// TwinCAT 3 PLC project SDSM3
// Title: SDS M2
// Company: Aperture Science
// Author: A. Wallace
// ProjectVersion: 2.6.1
// ProgramVersion: 3.1.0.9
// libraries:
//   LCLSVacuumLib, * (SLAC)
//   Tc2_Standard, * (Beckhoff Automation GmbH)
//   Tc2_System, * (Beckhoff Automation GmbH)
//   Tc3_Module, * (Beckhoff Automation GmbH)
//   LCLS General,0.1.2,SLAC
//   Tc2_EtherCAT,3.3.7.0,Beckhoff Automation GmbH
//   Tc2_IoFunctions,3.3.8.0,Beckhoff Automation GmbH
//   Tc2_MC2,3.3.15.0,Beckhoff Automation GmbH
//   Tc2_ModbusSrv,3.3.1.0,Beckhoff Automation GmbH
//   Tc2_SerialCom,3.3.6.0,Beckhoff Automation GmbH
//   Tc2_SUPS,3.3.4.0,Beckhoff Automation GmbH
//   Tc2_Utilities,3.3.17.0,Beckhoff Automation GmbH
// project tree:
//   DUTs/ALI/ E_AxisMoveMode.TcDUT (not stored), E_CTRL_MODE.TcDUT, E_PropValveFBState.TcDUT (not stored), HMI_PropValveCtrlState.TcDUT, ST_ALI.TcDUT, ST_ManipAxis.TcDUT, ST_PIDParams.TcDUT, ST_PressureController.TcDUT, ST_PropValveMKS253.TcDUT
//   DUTs/Bronkhorst/ E_BHElFlowUnit.TcDUT (not stored), ST_BhElFlow.TcDUT, ST_BhFMControl.TcDUT, ST_BhFMStatus.TcDUT
//   DUTs/ E_AxisMotionState.TcDUT, ST_M3GasManifold.TcDUT, ST_ManifoldValve.TcDUT (not stored), ST_Proportionair.TcDUT, ST_RegDeadbandControls.TcDUT (not stored), ST_Regulator.TcDUT (not stored), ST_Selector.TcDUT, ST_SelectorM3.TcDUT (not stored), ST_SensirionFM.TcDUT (not stored), ST_Shaker.TcDUT (not stored), ST_ShakerControls.TcDUT
//   DUTs/IO_Structs/ ST_ALIIO.TcDUT, ST_M2SelectorIO.TcDUT, ST_M3DeviceBaseIO.TcDUT (not stored), ST_M3GasManifoldIO.TcDUT (not stored), ST_M3PressCtrlIO.TcDUT (not stored), ST_M3SelectorIO.TcDUT
//   DUTs/Sensirion/ ST_SensirionFMControl.TcDUT, ST_SensirionFMStatus.TcDUT
//   DUTs/TEC/ ST_TECControl.TcDUT (not stored), ST_TECStatus.TcDUT (not stored)
//   DUTs/Vici/ ST_ViciControl.TcDUT, ST_ViciStatus.TcDUT (not stored)
//   GVLs/ GVL.TcGVL, GVL_Autosave.TcGVL, GVL_ComBuffers.TcGVL, GVL_Devices.TcGVL, GVL_IO.TcGVL, GVL_misc.TcGVL (not stored)
//   / PlcTask.TcTTO, SerialComm.TcTTO (not stored)
//   POUs/ALI/ FB_ALI.TcPOU, FB_PID_EXT.TcPOU, MC_SmoothMover.TcPOU, F_AxisRef_To_MSTA.TcPOU, FB_ManipAxis.TcPOU, FB_PropValve.TcPOU
//   POUs/Bronkhorst/ FB_L01Driver.TcPOU, FB_FlowBusTransaction.TcPOU (not stored)
//   POUs/ FB_SelectorM3.TcPOU, MAIN.TcPOU, p_ALI.TcPOU, p_Autosave.TcPOU, p_AutoWash.TcPOU, p_CoolerShaker.TcPOU, p_ESTOP.TcPOU, p_Manifold.TcPOU, p_ModbusRx.TcPOU, p_ModbusTx.TcPOU, p_Regulators.TcPOU, p_SampleSelector.TcPOU (not stored), p_SampleSelector2.TcPOU (not stored), p_Shakers.TcPOU, p_SoftIO.TcPOU, p_VacGaugeSup.TcPOU, SerialTxRx.TcPOU, p_StatusLights.TcPOU
//   POUs/Helpers/ FB_EcatDiag.TcPOU (not stored), FB_ManiValve.TcPOU (not stored), FB_SelectorSync.TcPOU, FB_ShiftByteArray.TcPOU
//   POUs/Regulators/ FB_ProportionairRegulator.TcPOU, FB_Regulator.TcPOU, F_rPressure.TcPOU (not stored)
//   POUs/Sensirion/ FB_SensirionDriver.TcPOU, FB_SensirionTransaction.TcPOU (not stored), fSHDLCChecksum.TcPOU (not stored)
//   POUs/TEC/ FB_TECDriver.TcPOU, FB_TECTransaction.TcPOU (not stored)
//   POUs/VICI/ FB_ViciDriver.TcPOU, FB_ViciTransaction.TcPOU
//   Version/ Global_Version.TcGVL
//   VISUs/ Main.TcVIS (not stored)
// real-time tasks:
//   TASK SerialComm: cycle T#5ms, priority 1, ADS port 350
//   TASK PlcTask: cycle T#10ms, priority 20, ADS port 351
// motion (NC):
//   TASK NC-Task 1 SAF: cycle T#2ms, priority 4, ADS port 501
//   TASK NC-Task 1 SVB: cycle T#10ms, priority 8, ADS port 511
//   AXIS ALI_X (id 3)
//     Dynamic: AccelerationMaximum=300, DecelerationMaximum=300, Acceleration=100, Deceleration=100
//     Velo: Maximum=5
//     PositionAreaControl: Range=0.005, RefSync=0.005
//     TargetPosControl: Range=0.0001
//     OtherSettings: AllowMotionCmdToSlave=true
//     encoder EncType=4
//       EncPara: ScaleFactorNumerator=0.001, MaxCount=#x0000ffff
//         Inc: RefSoftSyncMask=#x0000ffff
//     drive DrvType=24
//       Analog: VeloReferenz=12.7
//       TimeComp: TaskDelayCycles=1
//     controller CtrType=1
//       CtrPara: PriorControlFactor=1
//         PosDiffControl: Range=1
//         Observer: BandWidth=20
//   AXIS ALI_Z (id 5)
//     Dynamic: AccelerationMaximum=1000, DecelerationMaximum=1000, Acceleration=10, Deceleration=10, Jerk=100, DelayTime=0.08
//     Velo: Maximum=1
//     OtherSettings: AllowMotionCmdToSlave=true
//     encoder EncType=4
//       EncPara: ScaleFactorNumerator=3.96875e-005, MaxCount=#x0000ffff
//         Inc: RefSoftSyncMask=#x0000ffff
//     drive DrvType=24
//       Analog: VeloReferenz=5.08
//       TimeComp: TaskDelayCycles=1
//     controller CtrType=1
//       CtrPara: PriorControlFactor=1
//         PosDiffControl: Enable=false
//         Observer: BandWidth=20
//   AXIS ALI_Y (id 4)
//     Dynamic: DelayTime=0.08
//     Velo: Maximum=5
//     PositionAreaControl: Range=0.005, RefSync=0.005
//     TargetPosControl: Range=0.0001
//     OtherSettings: AllowMotionCmdToSlave=true
//     encoder EncType=4
//       EncPara: ScaleFactorNumerator=0.001, MaxCount=#x0000ffff
//         Inc: RefSoftSyncMask=#x0000ffff
//     drive DrvType=24
//       Analog: VeloReferenz=12.7
//       TimeComp: TaskDelayCycles=1
//     controller CtrType=1
//       CtrPara: PriorControlFactor=1
//         PosDiffControl: Range=1.5
//         Observer: BandWidth=20
//   AXIS ALI_PropValve (id 6)
//     General: UnitName=°
//     OtherSettings: AllowMotionCmdToSlave=true
//     encoder EncType=4
//       EncPara: ScaleFactorNumerator=0.028125, MaxCount=#x0000ffff
//         SoftEndMinControl: Enable=true
//         SoftEndMaxControl: Enable=true, Range=2900
//         Inc: RefSoftSyncMask=#x0000ffff
//     drive DrvType=24
//       Analog: VeloReferenz=3600
//       TimeComp: TaskDelayCycles=1
//     controller CtrType=1
//       CtrPara: PriorControlFactor=1
//         Observer: BandWidth=20
// I/O:
//   DEVICE MAIN (EtherCAT), AmsNetId 5.35.66.22.2.1
//     Term 1 (EK1200) [EK1200-5000 EtherCAT Power supply (2A E-Bus)]
//       Term 14 (EL3064) [EL3064 4Ch. Ana. Input 0-10V] (disabled)
//       Term 23 (EL4004) [EL4004 4Ch. Ana. Output 0-10V, 12bit] (disabled)
//       Term 25 (EL1124) [EL1124 4Ch. Dig. Input 5V, 10µs, Sensor Power] (disabled)
//       Term 17 (EL1008) [EL1008 8Ch. Dig. Input 24V, 3ms] (disabled)
//       Term 18 (EL2008) [EL2008 8Ch. Dig. Output 24V, 0.5A] (disabled)
//       Term 19 (EL2798) [EL2798 8Ch. Dig. Output 24V AC/DC, 2A, potential-free] (disabled)
//       Term 24 (EK1110) [EK1110 EtherCAT extension]
//     SC2 (EP9128-0021) [EP9128-0021 8x EtherCAT junction]
//       Box 32 (EP9128-1021) [EP9128-1021 8x EtherCAT junction - Dev A]
//       Box 33 (EP9128-2021) [EP9128-2021 8x EtherCAT junction - Dev B]
//     SC1 (EP9128-0021) [EP9128-0021 8x EtherCAT junction] (disabled)
//       Box 29 (EP9128-1021) [EP9128-1021 8x EtherCAT junction - Dev A]
//       Box 30 (EP9128-2021) [EP9128-2021 8x EtherCAT junction - Dev B]
//     SC3 (EP9128-0021) [EP9128-0021 8x EtherCAT junction] (disabled)
//       Box 21 (EP9128-1021) [EP9128-1021 8x EtherCAT junction - Dev A]
//       Box 22 (EP9128-2021) [EP9128-2021 8x EtherCAT junction - Dev B]
//     ALI (EP1111) [EP1111-0000 ID-Switch]
//     ALI_X (EP7041-0002) [EP7041-0002 1Ch. Stepper motor output stage (50V, 5A)]
//     ALI_Y (EP7041-0002) [EP7041-0002 1Ch. Stepper motor output stage (50V, 5A)]
//     ALI_Z (EP7041-0002) [EP7041-0002 1Ch. Stepper motor output stage (50V, 5A)]
//     ALI_X_ENC (EP5101-0011) [EP5101-0011 1Ch. Inc. Encoder 5V, D-SUB15]
//     ALI_Gauges (EP3174-0002) [EP3174-0002 4Ch. Ana. Input +/-10V, 0-10V, 0/4-20mA configurable]
//     ALI_PropValve (EP7041-0002) [EP7041-0002 1Ch. Stepper motor output stage (50V, 5A)]
//     ALI_Y_ENC (EP5101-0011) [EP5101-0011 1Ch. Inc. Encoder 5V, D-SUB15]
//     ALI_DIO (EP2338-0001) [EP2338-0001 8 Ch. Dig. Input/Output 24V, 0,5A, M8] (disabled)
//     M2 Selector A (EP1111) [EP1111-0000 ID-Switch]
//     M2 Selector A (EP6002-0002) [EP6002-0002 Interface (RS232/422/485)]
//     M2 Selector A (EP2338-0001) [EP2338-0001 8 Ch. Dig. Input/Output 24V, 0,5A, M8]
//     M2 Selector B (EP1111) [EP1111-0000 ID-Switch]
//     M2 Selector B (EP6002-0002) [EP6002-0002 Interface (RS232/422/485)]
//     M2 Selector B (EP2338-0001) [EP2338-0001 8 Ch. Dig. Input/Output 24V, 0,5A, M8]
//     M3 Selector A (EP1111) [EP1111-0000 ID-Switch]
//     M3 Selector A Digital IO (EP2338-1001) [EP2338-1001 8 Ch. Dig. Input/Output 24V, 3ms, 0,5A, M8]
//     M3 Selector A Serial IO (EP6002-0002) [EP6002-0002 Interface (RS232/422/485)]
//     M3 Selector A Mass Flow Meter (Mass Flow / Pressure Controller - Slave) [Mass Flow / Pressure Controller - Slave]
//     M3 Selector B (EP1111) [EP1111-0000 ID-Switch]
//     M3 Selector B Digital IO (EP2338-1001) [EP2338-1001 8 Ch. Dig. Input/Output 24V, 3ms, 0,5A, M8]
//     M3 Selector B Serial IO (EP6002-0002) [EP6002-0002 Interface (RS232/422/485)]
//     M3 Selector B Mass Flow Meter (Mass Flow / Pressure Controller - Slave) [Mass Flow / Pressure Controller - Slave]
//     PCM A (EP1111) [EP1111-0000 ID-Switch]
//     PCM A (EP4374-0002) [EP4374-0002 2Ch. Ana. Input +/-10V, 0-10V, 0/4-20mA configurable; 2Ch. Ana. Output +/-10V, 0-10V, 0/4-20mA configurable]
//     PCM A (EP3174-0002) [EP3174-0002 4Ch. Ana. Input +/-10V, 0-10V, 0/4-20mA configurable]
//     PCM A (EP6002-0002) [EP6002-0002 Interface (RS232/422/485)]
//     PCM B (EP1111) [EP1111-0000 ID-Switch]
//     PCM B (EP4374-0002) [EP4374-0002 2Ch. Ana. Input +/-10V, 0-10V, 0/4-20mA configurable; 2Ch. Ana. Output +/-10V, 0-10V, 0/4-20mA configurable]
//     PCM B (EP3174-0002) [EP3174-0002 4Ch. Ana. Input +/-10V, 0-10V, 0/4-20mA configurable] (disabled)
//     PCM B (EP6002-0002) [EP6002-0002 Interface (RS232/422/485)] (disabled)
//     Gas_Mani (EP1111) [EP1111-0000 ID-Switch]
//     Gas_Mani_NeedleValve (EP4374-0002) [EP4374-0002 2Ch. Ana. Input +/-10V, 0-10V, 0/4-20mA configurable; 2Ch. Ana. Output +/-10V, 0-10V, 0/4-20mA configurable]
//     Gas_Mani_ValveCtrl (EP2338-0001) [EP2338-0001 8 Ch. Dig. Input/Output 24V, 0,5A, M8]
//     Gas_Mani_ValveRbk (EP2338-0001) [EP2338-0001 8 Ch. Dig. Input/Output 24V, 0,5A, M8]
// variable links:
//   NC-Task 1 SAF/Axes/ALI_PropValve <-> MAIN (EtherCAT)/ALI_PropValve (EP7041-0002)
//     Drive/Inputs/In/nState1 @bit 3 <-> STM Status/Status/Error
//     Drive/Inputs/In/nState1 @bit 5 <-> STM Status/Status/Moving negative
//     Drive/Inputs/In/nState1 @bit 4 <-> STM Status/Status/Moving positive
//     Drive/Inputs/In/nState1 @bit 1 <-> STM Status/Status/Ready
//     Drive/Inputs/In/nState1 <-> STM Status/Status/Ready to enable
//     Drive/Inputs/In/nState1 @bit 6 <-> STM Status/Status/Torque reduced
//     Drive/Inputs/In/nState1 @bit 2 <-> STM Status/Status/Warning
//     Drive/Inputs/In/nState2 @bit 3 <-> STM Status/Status/Digital input 1
//     Drive/Inputs/In/nState2 @bit 4 <-> STM Status/Status/Digital input 2
//     Drive/Inputs/In/nState2 @bit 5 <-> STM Status/Status/Sync error
//     Drive/Inputs/In/nState2 @bit 7 <-> STM Status/Status/TxPDO Toggle
//     Drive/Inputs/In/nState4 @bit 1 <-> WcState/InputToggle
//     Drive/Inputs/In/nState4 <-> WcState/WcState
//     Drive/Outputs/Out/nCtrl1 <-> STM Control/Control/Enable
//     Drive/Outputs/Out/nCtrl1 @bit 2 <-> STM Control/Control/Reduce torque
//     Drive/Outputs/Out/nCtrl1 @bit 1 <-> STM Control/Control/Reset
//     Drive/Outputs/Out/nCtrl2 @bit 3 <-> STM Control/Control/Digital output 1
//     Drive/Outputs/Out/nDataOut2[0] <-> STM Velocity/Velocity
//     Enc/Inputs/In/nDataIn1[0] <-> ENC Status compact/Counter value
//     Enc/Inputs/In/nDataIn2[0] <-> ENC Status compact/Latch value
//     Enc/Inputs/In/nState1 @bit 4 <-> ENC Status compact/Status/Counter overflow
//     Enc/Inputs/In/nState1 @bit 3 <-> ENC Status compact/Status/Counter underflow
//     Enc/Inputs/In/nState1 @bit 7 <-> ENC Status compact/Status/Extrapolation stall
//     Enc/Inputs/In/nState1 <-> ENC Status compact/Status/Latch C valid
//     Enc/Inputs/In/nState1 @bit 1 <-> ENC Status compact/Status/Latch extern valid
//     Enc/Inputs/In/nState1 @bit 2 <-> ENC Status compact/Status/Set counter done
//     Enc/Inputs/In/nState2 @bit 4 <-> ENC Status compact/Status/Status of extern latch
//     Enc/Inputs/In/nState2 <-> ENC Status compact/Status/Status of input A
//     Enc/Inputs/In/nState2 @bit 1 <-> ENC Status compact/Status/Status of input B
//     Enc/Inputs/In/nState2 @bit 2 <-> ENC Status compact/Status/Status of input C
//     Enc/Inputs/In/nState2 @bit 5 <-> ENC Status compact/Status/Sync error
//     Enc/Inputs/In/nState2 @bit 7 <-> ENC Status compact/Status/TxPDO Toggle
//     Enc/Inputs/In/nState4 @bit 1 <-> WcState/InputToggle
//     Enc/Inputs/In/nState4 <-> WcState/WcState
//     Enc/Outputs/Out/nCtrl1 <-> ENC Control compact/Control/Enable latch C
//     Enc/Outputs/Out/nCtrl1 @bit 3 <-> ENC Control compact/Control/Enable latch extern on negative edge
//     Enc/Outputs/Out/nCtrl1 @bit 1 <-> ENC Control compact/Control/Enable latch extern on positive edge
//     Enc/Outputs/Out/nCtrl1 @bit 2 <-> ENC Control compact/Control/Set counter
//     Enc/Outputs/Out/nDataOut1[0] <-> ENC Control compact/Set counter value
//   NC-Task 1 SAF/Axes/ALI_X <-> MAIN (EtherCAT)/ALI_X (EP7041-0002)
//     Drive/Inputs/In/nState1 @bit 3 <-> STM Status/Status/Error
//     Drive/Inputs/In/nState1 @bit 5 <-> STM Status/Status/Moving negative
//     Drive/Inputs/In/nState1 @bit 4 <-> STM Status/Status/Moving positive
//     Drive/Inputs/In/nState1 @bit 1 <-> STM Status/Status/Ready
//     Drive/Inputs/In/nState1 <-> STM Status/Status/Ready to enable
//     Drive/Inputs/In/nState1 @bit 6 <-> STM Status/Status/Torque reduced
//     Drive/Inputs/In/nState1 @bit 2 <-> STM Status/Status/Warning
//     Drive/Inputs/In/nState2 @bit 3 <-> STM Status/Status/Digital input 1
//     Drive/Inputs/In/nState2 @bit 4 <-> STM Status/Status/Digital input 2
//     Drive/Inputs/In/nState2 @bit 5 <-> STM Status/Status/Sync error
//     Drive/Inputs/In/nState2 @bit 7 <-> STM Status/Status/TxPDO Toggle
//     Drive/Inputs/In/nState4 @bit 1 <-> WcState/InputToggle
//     Drive/Inputs/In/nState4 <-> WcState/WcState
//     Drive/Outputs/Out/nCtrl1 <-> STM Control/Control/Enable
//     Drive/Outputs/Out/nCtrl1 @bit 2 <-> STM Control/Control/Reduce torque
//     Drive/Outputs/Out/nCtrl1 @bit 1 <-> STM Control/Control/Reset
//     Drive/Outputs/Out/nCtrl2 @bit 3 <-> STM Control/Control/Digital output 1
//     Drive/Outputs/Out/nDataOut2[0] <-> STM Velocity/Velocity
//   NC-Task 1 SAF/Axes/ALI_X <-> MAIN (EtherCAT)/ALI_X_ENC (EP5101-0011)
//     Enc/Inputs/In/nDataIn1[0] <-> ENC Status compact/Counter value
//     Enc/Inputs/In/nDataIn2[0] <-> ENC Status compact/Latch value
//     Enc/Inputs/In/nState1 @bit 4 <-> ENC Status compact/Status/Counter overflow
//     Enc/Inputs/In/nState1 @bit 3 <-> ENC Status compact/Status/Counter underflow
//     Enc/Inputs/In/nState1 @bit 7 <-> ENC Status compact/Status/Extrapolation stall
//     Enc/Inputs/In/nState1 <-> ENC Status compact/Status/Latch C valid
//     Enc/Inputs/In/nState1 @bit 1 <-> ENC Status compact/Status/Latch extern valid
//     Enc/Inputs/In/nState1 @bit 6 <-> ENC Status compact/Status/Open circuit
//     Enc/Inputs/In/nState1 @bit 2 <-> ENC Status compact/Status/Set counter done
//     Enc/Inputs/In/nState1 @bit 5 <-> ENC Status compact/Status/Status of input status
//     Enc/Inputs/In/nState2 @bit 4 <-> ENC Status compact/Status/Status of extern latch
//     Enc/Inputs/In/nState2 <-> ENC Status compact/Status/Status of input A
//     Enc/Inputs/In/nState2 @bit 1 <-> ENC Status compact/Status/Status of input B
//     Enc/Inputs/In/nState2 @bit 2 <-> ENC Status compact/Status/Status of input C
//     Enc/Inputs/In/nState2 @bit 3 <-> ENC Status compact/Status/Status of input gate
//     Enc/Inputs/In/nState4 @bit 1 <-> WcState/InputToggle
//     Enc/Inputs/In/nState4 <-> WcState/WcState
//     Enc/Outputs/Out/nCtrl1 <-> ENC Control compact/Control/Enable latch C
//     Enc/Outputs/Out/nCtrl1 @bit 3 <-> ENC Control compact/Control/Enable latch extern on negative edge
//     Enc/Outputs/Out/nCtrl1 @bit 1 <-> ENC Control compact/Control/Enable latch extern on positive edge
//     Enc/Outputs/Out/nCtrl1 @bit 2 <-> ENC Control compact/Control/Set counter
//     Enc/Outputs/Out/nDataOut1[0] <-> ENC Control compact/Set counter value
//   NC-Task 1 SAF/Axes/ALI_Y <-> MAIN (EtherCAT)/ALI_Y (EP7041-0002)
//     Drive/Inputs/In/nState1 @bit 3 <-> STM Status/Status/Error
//     Drive/Inputs/In/nState1 @bit 5 <-> STM Status/Status/Moving negative
//     Drive/Inputs/In/nState1 @bit 4 <-> STM Status/Status/Moving positive
//     Drive/Inputs/In/nState1 @bit 1 <-> STM Status/Status/Ready
//     Drive/Inputs/In/nState1 <-> STM Status/Status/Ready to enable
//     Drive/Inputs/In/nState1 @bit 6 <-> STM Status/Status/Torque reduced
//     Drive/Inputs/In/nState1 @bit 2 <-> STM Status/Status/Warning
//     Drive/Inputs/In/nState2 @bit 3 <-> STM Status/Status/Digital input 1
//     Drive/Inputs/In/nState2 @bit 4 <-> STM Status/Status/Digital input 2
//     Drive/Inputs/In/nState2 @bit 5 <-> STM Status/Status/Sync error
//     Drive/Inputs/In/nState2 @bit 7 <-> STM Status/Status/TxPDO Toggle
//     Drive/Inputs/In/nState4 @bit 1 <-> WcState/InputToggle
//     Drive/Inputs/In/nState4 <-> WcState/WcState
//     Drive/Outputs/Out/nCtrl1 <-> STM Control/Control/Enable
//     Drive/Outputs/Out/nCtrl1 @bit 2 <-> STM Control/Control/Reduce torque
//     Drive/Outputs/Out/nCtrl1 @bit 1 <-> STM Control/Control/Reset
//     Drive/Outputs/Out/nCtrl2 @bit 3 <-> STM Control/Control/Digital output 1
//     Drive/Outputs/Out/nDataOut2[0] <-> STM Velocity/Velocity
//   NC-Task 1 SAF/Axes/ALI_Y <-> MAIN (EtherCAT)/ALI_Y_ENC (EP5101-0011)
//     Enc/Inputs/In/nDataIn1[0] <-> ENC Status compact/Counter value
//     Enc/Inputs/In/nDataIn2[0] <-> ENC Status compact/Latch value
//     Enc/Inputs/In/nState1 @bit 4 <-> ENC Status compact/Status/Counter overflow
//     Enc/Inputs/In/nState1 @bit 3 <-> ENC Status compact/Status/Counter underflow
//     Enc/Inputs/In/nState1 @bit 7 <-> ENC Status compact/Status/Extrapolation stall
//     Enc/Inputs/In/nState1 <-> ENC Status compact/Status/Latch C valid
//     Enc/Inputs/In/nState1 @bit 1 <-> ENC Status compact/Status/Latch extern valid
//     Enc/Inputs/In/nState1 @bit 6 <-> ENC Status compact/Status/Open circuit
//     Enc/Inputs/In/nState1 @bit 2 <-> ENC Status compact/Status/Set counter done
//     Enc/Inputs/In/nState1 @bit 5 <-> ENC Status compact/Status/Status of input status
//     Enc/Inputs/In/nState2 @bit 4 <-> ENC Status compact/Status/Status of extern latch
//     Enc/Inputs/In/nState2 <-> ENC Status compact/Status/Status of input A
//     Enc/Inputs/In/nState2 @bit 1 <-> ENC Status compact/Status/Status of input B
//     Enc/Inputs/In/nState2 @bit 2 <-> ENC Status compact/Status/Status of input C
//     Enc/Inputs/In/nState2 @bit 3 <-> ENC Status compact/Status/Status of input gate
//     Enc/Inputs/In/nState4 @bit 1 <-> WcState/InputToggle
//     Enc/Inputs/In/nState4 <-> WcState/WcState
//     Enc/Outputs/Out/nCtrl1 <-> ENC Control compact/Control/Enable latch C
//     Enc/Outputs/Out/nCtrl1 @bit 3 <-> ENC Control compact/Control/Enable latch extern on negative edge
//     Enc/Outputs/Out/nCtrl1 @bit 1 <-> ENC Control compact/Control/Enable latch extern on positive edge
//     Enc/Outputs/Out/nCtrl1 @bit 2 <-> ENC Control compact/Control/Set counter
//     Enc/Outputs/Out/nDataOut1[0] <-> ENC Control compact/Set counter value
//   NC-Task 1 SAF/Axes/ALI_Z <-> MAIN (EtherCAT)/ALI_Z (EP7041-0002)
//     Drive/Inputs/In/nState1 @bit 3 <-> STM Status/Status/Error
//     Drive/Inputs/In/nState1 @bit 5 <-> STM Status/Status/Moving negative
//     Drive/Inputs/In/nState1 @bit 4 <-> STM Status/Status/Moving positive
//     Drive/Inputs/In/nState1 @bit 1 <-> STM Status/Status/Ready
//     Drive/Inputs/In/nState1 <-> STM Status/Status/Ready to enable
//     Drive/Inputs/In/nState1 @bit 6 <-> STM Status/Status/Torque reduced
//     Drive/Inputs/In/nState1 @bit 2 <-> STM Status/Status/Warning
//     Drive/Inputs/In/nState2 @bit 3 <-> STM Status/Status/Digital input 1
//     Drive/Inputs/In/nState2 @bit 4 <-> STM Status/Status/Digital input 2
//     Drive/Inputs/In/nState2 @bit 5 <-> STM Status/Status/Sync error
//     Drive/Inputs/In/nState2 @bit 7 <-> STM Status/Status/TxPDO Toggle
//     Drive/Inputs/In/nState4 @bit 1 <-> WcState/InputToggle
//     Drive/Inputs/In/nState4 <-> WcState/WcState
//     Drive/Outputs/Out/nCtrl1 <-> STM Control/Control/Enable
//     Drive/Outputs/Out/nCtrl1 @bit 2 <-> STM Control/Control/Reduce torque
//     Drive/Outputs/Out/nCtrl1 @bit 1 <-> STM Control/Control/Reset
//     Drive/Outputs/Out/nCtrl2 @bit 3 <-> STM Control/Control/Digital output 1
//     Drive/Outputs/Out/nDataOut2[0] <-> STM Velocity/Velocity
//     Enc/Inputs/In/nDataIn1[0] <-> ENC Status compact/Counter value
//     Enc/Inputs/In/nDataIn2[0] <-> ENC Status compact/Latch value
//     Enc/Inputs/In/nState1 @bit 4 <-> ENC Status compact/Status/Counter overflow
//     Enc/Inputs/In/nState1 @bit 3 <-> ENC Status compact/Status/Counter underflow
//     Enc/Inputs/In/nState1 @bit 7 <-> ENC Status compact/Status/Extrapolation stall
//     Enc/Inputs/In/nState1 <-> ENC Status compact/Status/Latch C valid
//     Enc/Inputs/In/nState1 @bit 1 <-> ENC Status compact/Status/Latch extern valid
//     Enc/Inputs/In/nState1 @bit 2 <-> ENC Status compact/Status/Set counter done
//     Enc/Inputs/In/nState2 @bit 4 <-> ENC Status compact/Status/Status of extern latch
//     Enc/Inputs/In/nState2 <-> ENC Status compact/Status/Status of input A
//     Enc/Inputs/In/nState2 @bit 1 <-> ENC Status compact/Status/Status of input B
//     Enc/Inputs/In/nState2 @bit 2 <-> ENC Status compact/Status/Status of input C
//     Enc/Inputs/In/nState2 @bit 5 <-> ENC Status compact/Status/Sync error
//     Enc/Inputs/In/nState2 @bit 7 <-> ENC Status compact/Status/TxPDO Toggle
//     Enc/Inputs/In/nState4 @bit 1 <-> WcState/InputToggle
//     Enc/Inputs/In/nState4 <-> WcState/WcState
//     Enc/Outputs/Out/nCtrl1 <-> ENC Control compact/Control/Enable latch C
//     Enc/Outputs/Out/nCtrl1 @bit 3 <-> ENC Control compact/Control/Enable latch extern on negative edge
//     Enc/Outputs/Out/nCtrl1 @bit 1 <-> ENC Control compact/Control/Enable latch extern on positive edge
//     Enc/Outputs/Out/nCtrl1 @bit 2 <-> ENC Control compact/Control/Set counter
//     Enc/Outputs/Out/nDataOut1[0] <-> ENC Control compact/Set counter value
//   SDSM3/SDSM3 Instance <-> MAIN (EtherCAT)
//     PlcTask Inputs/GVL.g_aEcatMaster1 <-> InfoData/AmsNetId
//     PlcTask Inputs/GVL_Devices.stALI.i_SyncUnitWC <-> SyncUnits/[ALI (EP1111)]/PlcTask/WcState/WcState
//     PlcTask Inputs/GVL_IO.iq_stM2SelectorA.i_SyncUnitWC <-> SyncUnits/[M2 Selector A (EP1111)]/PlcTask/WcState/WcState
//     PlcTask Inputs/GVL_IO.iq_stM3SelectorA.i_SyncUnitWC <-> SyncUnits/[M3 Selector A (EP1111)]/PlcTask/WcState/WcState
//     PlcTask Inputs/GVL_IO.iq_stM2SelectorB.i_SyncUnitWC <-> SyncUnits/[M2 Selector B (EP1111)]/<unreferenced>/WcState/WcState
//     PlcTask Inputs/GVL_IO.iq_stM3GasManifold.i_SyncUnitWC <-> SyncUnits/[Gas_Mani (EP1111)]/PlcTask/WcState/WcState
//     PlcTask Inputs/GVL_IO.iq_stM3SelectorB.i_SyncUnitWC <-> SyncUnits/[M3 Selector B (EP1111)]/PlcTask/WcState/WcState
//     PlcTask Inputs/GVL_IO.iq_stPressCtrlA.i_SyncUnitWC <-> SyncUnits/[PCM A (EP1111)]/PlcTask/WcState/WcState
//     PlcTask Inputs/GVL_IO.iq_stPressCtrlB.i_SyncUnitWC <-> SyncUnits/[PCM B (EP1111)]/PlcTask/WcState/WcState
//   SDSM3/SDSM3 Instance <-> MAIN (EtherCAT)/ALI_Gauges (EP3174-0002)
//     PlcTask Inputs/GVL_Devices.stALI.i_EP3174_Ch{1..4} <-> AI Standard Channel {1..4}/Value  (4 links)
//   SDSM3/SDSM3 Instance <-> MAIN (EtherCAT)/ALI_PropValve (EP7041-0002)
//     PlcTask Inputs/GVL_Devices.stALI.stPropVlv.i_HLS <-> STM Status/Status/Digital input 1
//     PlcTask Inputs/GVL_Devices.stALI.stPropVlv.i_LLS <-> STM Status/Status/Digital input 2
//   SDSM3/SDSM3 Instance <-> MAIN (EtherCAT)/ALI_X (EP7041-0002)
//     PlcTask Inputs/GVL_Devices.stALI.axisX.xHiLS <-> STM Status/Status/Digital input 2
//     PlcTask Inputs/GVL_Devices.stALI.axisX.xLoLS <-> STM Status/Status/Digital input 1
//   SDSM3/SDSM3 Instance <-> MAIN (EtherCAT)/ALI_Y (EP7041-0002)
//     PlcTask Inputs/GVL_Devices.stALI.axisY.xHiLS <-> STM Status/Status/Digital input 2
//     PlcTask Inputs/GVL_Devices.stALI.axisY.xLoLS <-> STM Status/Status/Digital input 1
//   SDSM3/SDSM3 Instance <-> MAIN (EtherCAT)/ALI_Z (EP7041-0002)
//     PlcTask Inputs/GVL_Devices.stALI.axisZ.xHiLS <-> STM Status/Status/Digital input 2
//     PlcTask Inputs/GVL_Devices.stALI.axisZ.xLoLS <-> STM Status/Status/Digital input 1
//   SDSM3/SDSM3 Instance <-> MAIN (EtherCAT)/Gas_Mani_NeedleValve (EP4374-0002)
//     PlcTask Inputs/GVL_IO.iq_stM3GasManifold.i_EP4374_Ch1 <-> AI Inputs Channel 1/Value
//     PlcTask Inputs/GVL_IO.iq_stM3GasManifold.i_EP4374_Ch2 <-> AI Inputs Channel 2/Value
//     PlcTask Outputs/GVL_IO.iq_stM3GasManifold.q_EP4374_Ch3 <-> AO Outputs Channel 3/Analog output
//     PlcTask Outputs/GVL_IO.iq_stM3GasManifold.q_EP4374_Ch4 <-> AO Outputs Channel 4/Analog output
//   SDSM3/SDSM3 Instance <-> MAIN (EtherCAT)/Gas_Mani_ValveCtrl (EP2338-0001)
//     PlcTask Outputs/GVL_IO.iq_stM3GasManifold.q_EP2338_Ch{1..8} <-> Channel {9..16}/Output  (8 links)
//   SDSM3/SDSM3 Instance <-> MAIN (EtherCAT)/Gas_Mani_ValveRbk (EP2338-0001)
//     PlcTask Inputs/GVL_IO.iq_stM3GasManifold.i_EP2338_Ch{1..8} <-> Channel {1..8}/Input  (8 links)
//   SDSM3/SDSM3 Instance <-> MAIN (EtherCAT)/M2 Selector A (EP2338-0001)
//     PlcTask Inputs/GVL_IO.iq_stM2SelectorA.i_EP2338_Ch{5..8} <-> Channel {5..8}/Input  (4 links)
//     PlcTask Outputs/GVL_IO.iq_stM2SelectorA.q_EP2338_Ch{1..4} <-> Channel {9..12}/Output  (4 links)
//   SDSM3/SDSM3 Instance <-> MAIN (EtherCAT)/M2 Selector A (EP6002-0002)
//     SerialComm Inputs/GVL_IO.iq_stM2SelectorA.stComIn_EP6002P1/D[0] <-> COM TxPDO-Map Inputs Channel 1/Data In 0
//     SerialComm Inputs/GVL_IO.iq_stM2SelectorA.stComIn_EP6002P1/D[10] <-> COM TxPDO-Map Inputs Channel 1/Data In 10
//     SerialComm Inputs/GVL_IO.iq_stM2SelectorA.stComIn_EP6002P1/D[11] <-> COM TxPDO-Map Inputs Channel 1/Data In 11
//     SerialComm Inputs/GVL_IO.iq_stM2SelectorA.stComIn_EP6002P1/D[12] <-> COM TxPDO-Map Inputs Channel 1/Data In 12
//     SerialComm Inputs/GVL_IO.iq_stM2SelectorA.stComIn_EP6002P1/D[13] <-> COM TxPDO-Map Inputs Channel 1/Data In 13
//     SerialComm Inputs/GVL_IO.iq_stM2SelectorA.stComIn_EP6002P1/D[14] <-> COM TxPDO-Map Inputs Channel 1/Data In 14
//     SerialComm Inputs/GVL_IO.iq_stM2SelectorA.stComIn_EP6002P1/D[15] <-> COM TxPDO-Map Inputs Channel 1/Data In 15
//     SerialComm Inputs/GVL_IO.iq_stM2SelectorA.stComIn_EP6002P1/D[16] <-> COM TxPDO-Map Inputs Channel 1/Data In 16
//     SerialComm Inputs/GVL_IO.iq_stM2SelectorA.stComIn_EP6002P1/D[17] <-> COM TxPDO-Map Inputs Channel 1/Data In 17
//     SerialComm Inputs/GVL_IO.iq_stM2SelectorA.stComIn_EP6002P1/D[18] <-> COM TxPDO-Map Inputs Channel 1/Data In 18
//     SerialComm Inputs/GVL_IO.iq_stM2SelectorA.stComIn_EP6002P1/D[19] <-> COM TxPDO-Map Inputs Channel 1/Data In 19
//     SerialComm Inputs/GVL_IO.iq_stM2SelectorA.stComIn_EP6002P1/D[1] <-> COM TxPDO-Map Inputs Channel 1/Data In 1
//     SerialComm Inputs/GVL_IO.iq_stM2SelectorA.stComIn_EP6002P1/D[20] <-> COM TxPDO-Map Inputs Channel 1/Data In 20
//     SerialComm Inputs/GVL_IO.iq_stM2SelectorA.stComIn_EP6002P1/D[21] <-> COM TxPDO-Map Inputs Channel 1/Data In 21
//     SerialComm Inputs/GVL_IO.iq_stM2SelectorA.stComIn_EP6002P1/D[2] <-> COM TxPDO-Map Inputs Channel 1/Data In 2
//     SerialComm Inputs/GVL_IO.iq_stM2SelectorA.stComIn_EP6002P1/D[3] <-> COM TxPDO-Map Inputs Channel 1/Data In 3
//     SerialComm Inputs/GVL_IO.iq_stM2SelectorA.stComIn_EP6002P1/D[4] <-> COM TxPDO-Map Inputs Channel 1/Data In 4
//     SerialComm Inputs/GVL_IO.iq_stM2SelectorA.stComIn_EP6002P1/D[5] <-> COM TxPDO-Map Inputs Channel 1/Data In 5
//     SerialComm Inputs/GVL_IO.iq_stM2SelectorA.stComIn_EP6002P1/D[6] <-> COM TxPDO-Map Inputs Channel 1/Data In 6
//     SerialComm Inputs/GVL_IO.iq_stM2SelectorA.stComIn_EP6002P1/D[7] <-> COM TxPDO-Map Inputs Channel 1/Data In 7
//     SerialComm Inputs/GVL_IO.iq_stM2SelectorA.stComIn_EP6002P1/D[8] <-> COM TxPDO-Map Inputs Channel 1/Data In 8
//     SerialComm Inputs/GVL_IO.iq_stM2SelectorA.stComIn_EP6002P1/D[9] <-> COM TxPDO-Map Inputs Channel 1/Data In 9
//     SerialComm Inputs/GVL_IO.iq_stM2SelectorA.stComIn_EP6002P2/D[0] <-> COM TxPDO-Map Inputs Channel 2/Data In 0
//     SerialComm Inputs/GVL_IO.iq_stM2SelectorA.stComIn_EP6002P2/D[10] <-> COM TxPDO-Map Inputs Channel 2/Data In 10
//     SerialComm Inputs/GVL_IO.iq_stM2SelectorA.stComIn_EP6002P2/D[11] <-> COM TxPDO-Map Inputs Channel 2/Data In 11
//     SerialComm Inputs/GVL_IO.iq_stM2SelectorA.stComIn_EP6002P2/D[12] <-> COM TxPDO-Map Inputs Channel 2/Data In 12
//     SerialComm Inputs/GVL_IO.iq_stM2SelectorA.stComIn_EP6002P2/D[13] <-> COM TxPDO-Map Inputs Channel 2/Data In 13
//     SerialComm Inputs/GVL_IO.iq_stM2SelectorA.stComIn_EP6002P2/D[14] <-> COM TxPDO-Map Inputs Channel 2/Data In 14
//     SerialComm Inputs/GVL_IO.iq_stM2SelectorA.stComIn_EP6002P2/D[15] <-> COM TxPDO-Map Inputs Channel 2/Data In 15
//     SerialComm Inputs/GVL_IO.iq_stM2SelectorA.stComIn_EP6002P2/D[16] <-> COM TxPDO-Map Inputs Channel 2/Data In 16
//     SerialComm Inputs/GVL_IO.iq_stM2SelectorA.stComIn_EP6002P2/D[17] <-> COM TxPDO-Map Inputs Channel 2/Data In 17
//     SerialComm Inputs/GVL_IO.iq_stM2SelectorA.stComIn_EP6002P2/D[18] <-> COM TxPDO-Map Inputs Channel 2/Data In 18
//     SerialComm Inputs/GVL_IO.iq_stM2SelectorA.stComIn_EP6002P2/D[19] <-> COM TxPDO-Map Inputs Channel 2/Data In 19
//     SerialComm Inputs/GVL_IO.iq_stM2SelectorA.stComIn_EP6002P2/D[1] <-> COM TxPDO-Map Inputs Channel 2/Data In 1
//     SerialComm Inputs/GVL_IO.iq_stM2SelectorA.stComIn_EP6002P2/D[20] <-> COM TxPDO-Map Inputs Channel 2/Data In 20
//     SerialComm Inputs/GVL_IO.iq_stM2SelectorA.stComIn_EP6002P2/D[21] <-> COM TxPDO-Map Inputs Channel 2/Data In 21
//     SerialComm Inputs/GVL_IO.iq_stM2SelectorA.stComIn_EP6002P2/D[2] <-> COM TxPDO-Map Inputs Channel 2/Data In 2
//     SerialComm Inputs/GVL_IO.iq_stM2SelectorA.stComIn_EP6002P2/D[3] <-> COM TxPDO-Map Inputs Channel 2/Data In 3
//     SerialComm Inputs/GVL_IO.iq_stM2SelectorA.stComIn_EP6002P2/D[4] <-> COM TxPDO-Map Inputs Channel 2/Data In 4
//     SerialComm Inputs/GVL_IO.iq_stM2SelectorA.stComIn_EP6002P2/D[5] <-> COM TxPDO-Map Inputs Channel 2/Data In 5
//     SerialComm Inputs/GVL_IO.iq_stM2SelectorA.stComIn_EP6002P2/D[6] <-> COM TxPDO-Map Inputs Channel 2/Data In 6
//     SerialComm Inputs/GVL_IO.iq_stM2SelectorA.stComIn_EP6002P2/D[7] <-> COM TxPDO-Map Inputs Channel 2/Data In 7
//     SerialComm Inputs/GVL_IO.iq_stM2SelectorA.stComIn_EP6002P2/D[8] <-> COM TxPDO-Map Inputs Channel 2/Data In 8
//     SerialComm Inputs/GVL_IO.iq_stM2SelectorA.stComIn_EP6002P2/D[9] <-> COM TxPDO-Map Inputs Channel 2/Data In 9
//     SerialComm Inputs/GVL_IO.iq_stM2SelectorA.stComIn_EP6002P1/Status <-> COM TxPDO-Map Inputs Channel 1/Status
//     SerialComm Inputs/GVL_IO.iq_stM2SelectorA.stComIn_EP6002P2/Status <-> COM TxPDO-Map Inputs Channel 2/Status
//     SerialComm Outputs/GVL_IO.iq_stM2SelectorA.stComOut_EP6002P1/Ctrl <-> COM RxPDO-Map Outputs Channel 1/Ctrl
//     SerialComm Outputs/GVL_IO.iq_stM2SelectorA.stComOut_EP6002P2/Ctrl <-> COM RxPDO-Map Outputs Channel 2/Ctrl
//     SerialComm Outputs/GVL_IO.iq_stM2SelectorA.stComOut_EP6002P1/D[0] <-> COM RxPDO-Map Outputs Channel 1/Data Out 0
//     SerialComm Outputs/GVL_IO.iq_stM2SelectorA.stComOut_EP6002P1/D[10] <-> COM RxPDO-Map Outputs Channel 1/Data Out 10
//     SerialComm Outputs/GVL_IO.iq_stM2SelectorA.stComOut_EP6002P1/D[11] <-> COM RxPDO-Map Outputs Channel 1/Data Out 11
//     SerialComm Outputs/GVL_IO.iq_stM2SelectorA.stComOut_EP6002P1/D[12] <-> COM RxPDO-Map Outputs Channel 1/Data Out 12
//     SerialComm Outputs/GVL_IO.iq_stM2SelectorA.stComOut_EP6002P1/D[13] <-> COM RxPDO-Map Outputs Channel 1/Data Out 13
//     SerialComm Outputs/GVL_IO.iq_stM2SelectorA.stComOut_EP6002P1/D[14] <-> COM RxPDO-Map Outputs Channel 1/Data Out 14
//     SerialComm Outputs/GVL_IO.iq_stM2SelectorA.stComOut_EP6002P1/D[15] <-> COM RxPDO-Map Outputs Channel 1/Data Out 15
//     SerialComm Outputs/GVL_IO.iq_stM2SelectorA.stComOut_EP6002P1/D[16] <-> COM RxPDO-Map Outputs Channel 1/Data Out 16
//     SerialComm Outputs/GVL_IO.iq_stM2SelectorA.stComOut_EP6002P1/D[17] <-> COM RxPDO-Map Outputs Channel 1/Data Out 17
//     SerialComm Outputs/GVL_IO.iq_stM2SelectorA.stComOut_EP6002P1/D[18] <-> COM RxPDO-Map Outputs Channel 1/Data Out 18
//     SerialComm Outputs/GVL_IO.iq_stM2SelectorA.stComOut_EP6002P1/D[19] <-> COM RxPDO-Map Outputs Channel 1/Data Out 19
//     SerialComm Outputs/GVL_IO.iq_stM2SelectorA.stComOut_EP6002P1/D[1] <-> COM RxPDO-Map Outputs Channel 1/Data Out 1
//     SerialComm Outputs/GVL_IO.iq_stM2SelectorA.stComOut_EP6002P1/D[20] <-> COM RxPDO-Map Outputs Channel 1/Data Out 20
//     SerialComm Outputs/GVL_IO.iq_stM2SelectorA.stComOut_EP6002P1/D[21] <-> COM RxPDO-Map Outputs Channel 1/Data Out 21
//     SerialComm Outputs/GVL_IO.iq_stM2SelectorA.stComOut_EP6002P1/D[2] <-> COM RxPDO-Map Outputs Channel 1/Data Out 2
//     SerialComm Outputs/GVL_IO.iq_stM2SelectorA.stComOut_EP6002P1/D[3] <-> COM RxPDO-Map Outputs Channel 1/Data Out 3
//     SerialComm Outputs/GVL_IO.iq_stM2SelectorA.stComOut_EP6002P1/D[4] <-> COM RxPDO-Map Outputs Channel 1/Data Out 4
//     SerialComm Outputs/GVL_IO.iq_stM2SelectorA.stComOut_EP6002P1/D[5] <-> COM RxPDO-Map Outputs Channel 1/Data Out 5
//     SerialComm Outputs/GVL_IO.iq_stM2SelectorA.stComOut_EP6002P1/D[6] <-> COM RxPDO-Map Outputs Channel 1/Data Out 6
//     SerialComm Outputs/GVL_IO.iq_stM2SelectorA.stComOut_EP6002P1/D[7] <-> COM RxPDO-Map Outputs Channel 1/Data Out 7
//     SerialComm Outputs/GVL_IO.iq_stM2SelectorA.stComOut_EP6002P1/D[8] <-> COM RxPDO-Map Outputs Channel 1/Data Out 8
//     SerialComm Outputs/GVL_IO.iq_stM2SelectorA.stComOut_EP6002P1/D[9] <-> COM RxPDO-Map Outputs Channel 1/Data Out 9
//     SerialComm Outputs/GVL_IO.iq_stM2SelectorA.stComOut_EP6002P2/D[0] <-> COM RxPDO-Map Outputs Channel 2/Data Out 0
//     SerialComm Outputs/GVL_IO.iq_stM2SelectorA.stComOut_EP6002P2/D[10] <-> COM RxPDO-Map Outputs Channel 2/Data Out 10
//     SerialComm Outputs/GVL_IO.iq_stM2SelectorA.stComOut_EP6002P2/D[11] <-> COM RxPDO-Map Outputs Channel 2/Data Out 11
//     SerialComm Outputs/GVL_IO.iq_stM2SelectorA.stComOut_EP6002P2/D[12] <-> COM RxPDO-Map Outputs Channel 2/Data Out 12
//     SerialComm Outputs/GVL_IO.iq_stM2SelectorA.stComOut_EP6002P2/D[13] <-> COM RxPDO-Map Outputs Channel 2/Data Out 13
//     SerialComm Outputs/GVL_IO.iq_stM2SelectorA.stComOut_EP6002P2/D[14] <-> COM RxPDO-Map Outputs Channel 2/Data Out 14
//     SerialComm Outputs/GVL_IO.iq_stM2SelectorA.stComOut_EP6002P2/D[15] <-> COM RxPDO-Map Outputs Channel 2/Data Out 15
//     SerialComm Outputs/GVL_IO.iq_stM2SelectorA.stComOut_EP6002P2/D[16] <-> COM RxPDO-Map Outputs Channel 2/Data Out 16
//     SerialComm Outputs/GVL_IO.iq_stM2SelectorA.stComOut_EP6002P2/D[17] <-> COM RxPDO-Map Outputs Channel 2/Data Out 17
//     SerialComm Outputs/GVL_IO.iq_stM2SelectorA.stComOut_EP6002P2/D[18] <-> COM RxPDO-Map Outputs Channel 2/Data Out 18
//     SerialComm Outputs/GVL_IO.iq_stM2SelectorA.stComOut_EP6002P2/D[19] <-> COM RxPDO-Map Outputs Channel 2/Data Out 19
//     SerialComm Outputs/GVL_IO.iq_stM2SelectorA.stComOut_EP6002P2/D[1] <-> COM RxPDO-Map Outputs Channel 2/Data Out 1
//     SerialComm Outputs/GVL_IO.iq_stM2SelectorA.stComOut_EP6002P2/D[20] <-> COM RxPDO-Map Outputs Channel 2/Data Out 20
//     SerialComm Outputs/GVL_IO.iq_stM2SelectorA.stComOut_EP6002P2/D[21] <-> COM RxPDO-Map Outputs Channel 2/Data Out 21
//     SerialComm Outputs/GVL_IO.iq_stM2SelectorA.stComOut_EP6002P2/D[2] <-> COM RxPDO-Map Outputs Channel 2/Data Out 2
//     SerialComm Outputs/GVL_IO.iq_stM2SelectorA.stComOut_EP6002P2/D[3] <-> COM RxPDO-Map Outputs Channel 2/Data Out 3
//     SerialComm Outputs/GVL_IO.iq_stM2SelectorA.stComOut_EP6002P2/D[4] <-> COM RxPDO-Map Outputs Channel 2/Data Out 4
//     SerialComm Outputs/GVL_IO.iq_stM2SelectorA.stComOut_EP6002P2/D[5] <-> COM RxPDO-Map Outputs Channel 2/Data Out 5
//     SerialComm Outputs/GVL_IO.iq_stM2SelectorA.stComOut_EP6002P2/D[6] <-> COM RxPDO-Map Outputs Channel 2/Data Out 6
//     SerialComm Outputs/GVL_IO.iq_stM2SelectorA.stComOut_EP6002P2/D[7] <-> COM RxPDO-Map Outputs Channel 2/Data Out 7
//     SerialComm Outputs/GVL_IO.iq_stM2SelectorA.stComOut_EP6002P2/D[8] <-> COM RxPDO-Map Outputs Channel 2/Data Out 8
//     SerialComm Outputs/GVL_IO.iq_stM2SelectorA.stComOut_EP6002P2/D[9] <-> COM RxPDO-Map Outputs Channel 2/Data Out 9
//   SDSM3/SDSM3 Instance <-> MAIN (EtherCAT)/M2 Selector B (EP2338-0001)
//     PlcTask Inputs/GVL_IO.iq_stM2SelectorB.i_EP2338_Ch{5..8} <-> Channel {5..8}/Input  (4 links)
//     PlcTask Outputs/GVL_IO.iq_stM2SelectorB.q_EP2338_Ch{1..4} <-> Channel {9..12}/Output  (4 links)
//   SDSM3/SDSM3 Instance <-> MAIN (EtherCAT)/M2 Selector B (EP6002-0002)
//     SerialComm Inputs/GVL_IO.iq_stM2SelectorB.stComIn_EP6002P1/D[0] <-> COM TxPDO-Map Inputs Channel 1/Data In 0
//     SerialComm Inputs/GVL_IO.iq_stM2SelectorB.stComIn_EP6002P1/D[10] <-> COM TxPDO-Map Inputs Channel 1/Data In 10
//     SerialComm Inputs/GVL_IO.iq_stM2SelectorB.stComIn_EP6002P1/D[11] <-> COM TxPDO-Map Inputs Channel 1/Data In 11
//     SerialComm Inputs/GVL_IO.iq_stM2SelectorB.stComIn_EP6002P1/D[12] <-> COM TxPDO-Map Inputs Channel 1/Data In 12
//     SerialComm Inputs/GVL_IO.iq_stM2SelectorB.stComIn_EP6002P1/D[13] <-> COM TxPDO-Map Inputs Channel 1/Data In 13
//     SerialComm Inputs/GVL_IO.iq_stM2SelectorB.stComIn_EP6002P1/D[14] <-> COM TxPDO-Map Inputs Channel 1/Data In 14
//     SerialComm Inputs/GVL_IO.iq_stM2SelectorB.stComIn_EP6002P1/D[15] <-> COM TxPDO-Map Inputs Channel 1/Data In 15
//     SerialComm Inputs/GVL_IO.iq_stM2SelectorB.stComIn_EP6002P1/D[16] <-> COM TxPDO-Map Inputs Channel 1/Data In 16
//     SerialComm Inputs/GVL_IO.iq_stM2SelectorB.stComIn_EP6002P1/D[17] <-> COM TxPDO-Map Inputs Channel 1/Data In 17
//     SerialComm Inputs/GVL_IO.iq_stM2SelectorB.stComIn_EP6002P1/D[18] <-> COM TxPDO-Map Inputs Channel 1/Data In 18
//     SerialComm Inputs/GVL_IO.iq_stM2SelectorB.stComIn_EP6002P1/D[19] <-> COM TxPDO-Map Inputs Channel 1/Data In 19
//     SerialComm Inputs/GVL_IO.iq_stM2SelectorB.stComIn_EP6002P1/D[1] <-> COM TxPDO-Map Inputs Channel 1/Data In 1
//     SerialComm Inputs/GVL_IO.iq_stM2SelectorB.stComIn_EP6002P1/D[20] <-> COM TxPDO-Map Inputs Channel 1/Data In 20
//     SerialComm Inputs/GVL_IO.iq_stM2SelectorB.stComIn_EP6002P1/D[21] <-> COM TxPDO-Map Inputs Channel 1/Data In 21
//     SerialComm Inputs/GVL_IO.iq_stM2SelectorB.stComIn_EP6002P1/D[2] <-> COM TxPDO-Map Inputs Channel 1/Data In 2
//     SerialComm Inputs/GVL_IO.iq_stM2SelectorB.stComIn_EP6002P1/D[3] <-> COM TxPDO-Map Inputs Channel 1/Data In 3
//     SerialComm Inputs/GVL_IO.iq_stM2SelectorB.stComIn_EP6002P1/D[4] <-> COM TxPDO-Map Inputs Channel 1/Data In 4
//     SerialComm Inputs/GVL_IO.iq_stM2SelectorB.stComIn_EP6002P1/D[5] <-> COM TxPDO-Map Inputs Channel 1/Data In 5
//     SerialComm Inputs/GVL_IO.iq_stM2SelectorB.stComIn_EP6002P1/D[6] <-> COM TxPDO-Map Inputs Channel 1/Data In 6
//     SerialComm Inputs/GVL_IO.iq_stM2SelectorB.stComIn_EP6002P1/D[7] <-> COM TxPDO-Map Inputs Channel 1/Data In 7
//     SerialComm Inputs/GVL_IO.iq_stM2SelectorB.stComIn_EP6002P1/D[8] <-> COM TxPDO-Map Inputs Channel 1/Data In 8
//     SerialComm Inputs/GVL_IO.iq_stM2SelectorB.stComIn_EP6002P1/D[9] <-> COM TxPDO-Map Inputs Channel 1/Data In 9
//     SerialComm Inputs/GVL_IO.iq_stM2SelectorB.stComIn_EP6002P2/D[0] <-> COM TxPDO-Map Inputs Channel 2/Data In 0
//     SerialComm Inputs/GVL_IO.iq_stM2SelectorB.stComIn_EP6002P2/D[10] <-> COM TxPDO-Map Inputs Channel 2/Data In 10
//     SerialComm Inputs/GVL_IO.iq_stM2SelectorB.stComIn_EP6002P2/D[11] <-> COM TxPDO-Map Inputs Channel 2/Data In 11
//     SerialComm Inputs/GVL_IO.iq_stM2SelectorB.stComIn_EP6002P2/D[12] <-> COM TxPDO-Map Inputs Channel 2/Data In 12
//     SerialComm Inputs/GVL_IO.iq_stM2SelectorB.stComIn_EP6002P2/D[13] <-> COM TxPDO-Map Inputs Channel 2/Data In 13
//     SerialComm Inputs/GVL_IO.iq_stM2SelectorB.stComIn_EP6002P2/D[14] <-> COM TxPDO-Map Inputs Channel 2/Data In 14
//     SerialComm Inputs/GVL_IO.iq_stM2SelectorB.stComIn_EP6002P2/D[15] <-> COM TxPDO-Map Inputs Channel 2/Data In 15
//     SerialComm Inputs/GVL_IO.iq_stM2SelectorB.stComIn_EP6002P2/D[16] <-> COM TxPDO-Map Inputs Channel 2/Data In 16
//     SerialComm Inputs/GVL_IO.iq_stM2SelectorB.stComIn_EP6002P2/D[17] <-> COM TxPDO-Map Inputs Channel 2/Data In 17
//     SerialComm Inputs/GVL_IO.iq_stM2SelectorB.stComIn_EP6002P2/D[18] <-> COM TxPDO-Map Inputs Channel 2/Data In 18
//     SerialComm Inputs/GVL_IO.iq_stM2SelectorB.stComIn_EP6002P2/D[19] <-> COM TxPDO-Map Inputs Channel 2/Data In 19
//     SerialComm Inputs/GVL_IO.iq_stM2SelectorB.stComIn_EP6002P2/D[1] <-> COM TxPDO-Map Inputs Channel 2/Data In 1
//     SerialComm Inputs/GVL_IO.iq_stM2SelectorB.stComIn_EP6002P2/D[20] <-> COM TxPDO-Map Inputs Channel 2/Data In 20
//     SerialComm Inputs/GVL_IO.iq_stM2SelectorB.stComIn_EP6002P2/D[21] <-> COM TxPDO-Map Inputs Channel 2/Data In 21
//     SerialComm Inputs/GVL_IO.iq_stM2SelectorB.stComIn_EP6002P2/D[2] <-> COM TxPDO-Map Inputs Channel 2/Data In 2
//     SerialComm Inputs/GVL_IO.iq_stM2SelectorB.stComIn_EP6002P2/D[3] <-> COM TxPDO-Map Inputs Channel 2/Data In 3
//     SerialComm Inputs/GVL_IO.iq_stM2SelectorB.stComIn_EP6002P2/D[4] <-> COM TxPDO-Map Inputs Channel 2/Data In 4
//     SerialComm Inputs/GVL_IO.iq_stM2SelectorB.stComIn_EP6002P2/D[5] <-> COM TxPDO-Map Inputs Channel 2/Data In 5
//     SerialComm Inputs/GVL_IO.iq_stM2SelectorB.stComIn_EP6002P2/D[6] <-> COM TxPDO-Map Inputs Channel 2/Data In 6
//     SerialComm Inputs/GVL_IO.iq_stM2SelectorB.stComIn_EP6002P2/D[7] <-> COM TxPDO-Map Inputs Channel 2/Data In 7
//     SerialComm Inputs/GVL_IO.iq_stM2SelectorB.stComIn_EP6002P2/D[8] <-> COM TxPDO-Map Inputs Channel 2/Data In 8
//     SerialComm Inputs/GVL_IO.iq_stM2SelectorB.stComIn_EP6002P2/D[9] <-> COM TxPDO-Map Inputs Channel 2/Data In 9
//     SerialComm Inputs/GVL_IO.iq_stM2SelectorB.stComIn_EP6002P1/Status <-> COM TxPDO-Map Inputs Channel 1/Status
//     SerialComm Inputs/GVL_IO.iq_stM2SelectorB.stComIn_EP6002P2/Status <-> COM TxPDO-Map Inputs Channel 2/Status
//     SerialComm Outputs/GVL_IO.iq_stM2SelectorB.stComOut_EP6002P1/Ctrl <-> COM RxPDO-Map Outputs Channel 1/Ctrl
//     SerialComm Outputs/GVL_IO.iq_stM2SelectorB.stComOut_EP6002P2/Ctrl <-> COM RxPDO-Map Outputs Channel 2/Ctrl
//     SerialComm Outputs/GVL_IO.iq_stM2SelectorB.stComOut_EP6002P1/D[0] <-> COM RxPDO-Map Outputs Channel 1/Data Out 0
//     SerialComm Outputs/GVL_IO.iq_stM2SelectorB.stComOut_EP6002P1/D[10] <-> COM RxPDO-Map Outputs Channel 1/Data Out 10
//     SerialComm Outputs/GVL_IO.iq_stM2SelectorB.stComOut_EP6002P1/D[11] <-> COM RxPDO-Map Outputs Channel 1/Data Out 11
//     SerialComm Outputs/GVL_IO.iq_stM2SelectorB.stComOut_EP6002P1/D[12] <-> COM RxPDO-Map Outputs Channel 1/Data Out 12
//     SerialComm Outputs/GVL_IO.iq_stM2SelectorB.stComOut_EP6002P1/D[13] <-> COM RxPDO-Map Outputs Channel 1/Data Out 13
//     SerialComm Outputs/GVL_IO.iq_stM2SelectorB.stComOut_EP6002P1/D[14] <-> COM RxPDO-Map Outputs Channel 1/Data Out 14
//     SerialComm Outputs/GVL_IO.iq_stM2SelectorB.stComOut_EP6002P1/D[15] <-> COM RxPDO-Map Outputs Channel 1/Data Out 15
//     SerialComm Outputs/GVL_IO.iq_stM2SelectorB.stComOut_EP6002P1/D[16] <-> COM RxPDO-Map Outputs Channel 1/Data Out 16
//     SerialComm Outputs/GVL_IO.iq_stM2SelectorB.stComOut_EP6002P1/D[17] <-> COM RxPDO-Map Outputs Channel 1/Data Out 17
//     SerialComm Outputs/GVL_IO.iq_stM2SelectorB.stComOut_EP6002P1/D[18] <-> COM RxPDO-Map Outputs Channel 1/Data Out 18
//     SerialComm Outputs/GVL_IO.iq_stM2SelectorB.stComOut_EP6002P1/D[19] <-> COM RxPDO-Map Outputs Channel 1/Data Out 19
//     SerialComm Outputs/GVL_IO.iq_stM2SelectorB.stComOut_EP6002P1/D[1] <-> COM RxPDO-Map Outputs Channel 1/Data Out 1
//     SerialComm Outputs/GVL_IO.iq_stM2SelectorB.stComOut_EP6002P1/D[20] <-> COM RxPDO-Map Outputs Channel 1/Data Out 20
//     SerialComm Outputs/GVL_IO.iq_stM2SelectorB.stComOut_EP6002P1/D[21] <-> COM RxPDO-Map Outputs Channel 1/Data Out 21
//     SerialComm Outputs/GVL_IO.iq_stM2SelectorB.stComOut_EP6002P1/D[2] <-> COM RxPDO-Map Outputs Channel 1/Data Out 2
//     SerialComm Outputs/GVL_IO.iq_stM2SelectorB.stComOut_EP6002P1/D[3] <-> COM RxPDO-Map Outputs Channel 1/Data Out 3
//     SerialComm Outputs/GVL_IO.iq_stM2SelectorB.stComOut_EP6002P1/D[4] <-> COM RxPDO-Map Outputs Channel 1/Data Out 4
//     SerialComm Outputs/GVL_IO.iq_stM2SelectorB.stComOut_EP6002P1/D[5] <-> COM RxPDO-Map Outputs Channel 1/Data Out 5
//     SerialComm Outputs/GVL_IO.iq_stM2SelectorB.stComOut_EP6002P1/D[6] <-> COM RxPDO-Map Outputs Channel 1/Data Out 6
//     SerialComm Outputs/GVL_IO.iq_stM2SelectorB.stComOut_EP6002P1/D[7] <-> COM RxPDO-Map Outputs Channel 1/Data Out 7
//     SerialComm Outputs/GVL_IO.iq_stM2SelectorB.stComOut_EP6002P1/D[8] <-> COM RxPDO-Map Outputs Channel 1/Data Out 8
//     SerialComm Outputs/GVL_IO.iq_stM2SelectorB.stComOut_EP6002P1/D[9] <-> COM RxPDO-Map Outputs Channel 1/Data Out 9
//     SerialComm Outputs/GVL_IO.iq_stM2SelectorB.stComOut_EP6002P2/D[0] <-> COM RxPDO-Map Outputs Channel 2/Data Out 0
//     SerialComm Outputs/GVL_IO.iq_stM2SelectorB.stComOut_EP6002P2/D[10] <-> COM RxPDO-Map Outputs Channel 2/Data Out 10
//     SerialComm Outputs/GVL_IO.iq_stM2SelectorB.stComOut_EP6002P2/D[11] <-> COM RxPDO-Map Outputs Channel 2/Data Out 11
//     SerialComm Outputs/GVL_IO.iq_stM2SelectorB.stComOut_EP6002P2/D[12] <-> COM RxPDO-Map Outputs Channel 2/Data Out 12
//     SerialComm Outputs/GVL_IO.iq_stM2SelectorB.stComOut_EP6002P2/D[13] <-> COM RxPDO-Map Outputs Channel 2/Data Out 13
//     SerialComm Outputs/GVL_IO.iq_stM2SelectorB.stComOut_EP6002P2/D[14] <-> COM RxPDO-Map Outputs Channel 2/Data Out 14
//     SerialComm Outputs/GVL_IO.iq_stM2SelectorB.stComOut_EP6002P2/D[15] <-> COM RxPDO-Map Outputs Channel 2/Data Out 15
//     SerialComm Outputs/GVL_IO.iq_stM2SelectorB.stComOut_EP6002P2/D[16] <-> COM RxPDO-Map Outputs Channel 2/Data Out 16
//     SerialComm Outputs/GVL_IO.iq_stM2SelectorB.stComOut_EP6002P2/D[17] <-> COM RxPDO-Map Outputs Channel 2/Data Out 17
//     SerialComm Outputs/GVL_IO.iq_stM2SelectorB.stComOut_EP6002P2/D[18] <-> COM RxPDO-Map Outputs Channel 2/Data Out 18
//     SerialComm Outputs/GVL_IO.iq_stM2SelectorB.stComOut_EP6002P2/D[19] <-> COM RxPDO-Map Outputs Channel 2/Data Out 19
//     SerialComm Outputs/GVL_IO.iq_stM2SelectorB.stComOut_EP6002P2/D[1] <-> COM RxPDO-Map Outputs Channel 2/Data Out 1
//     SerialComm Outputs/GVL_IO.iq_stM2SelectorB.stComOut_EP6002P2/D[20] <-> COM RxPDO-Map Outputs Channel 2/Data Out 20
//     SerialComm Outputs/GVL_IO.iq_stM2SelectorB.stComOut_EP6002P2/D[21] <-> COM RxPDO-Map Outputs Channel 2/Data Out 21
//     SerialComm Outputs/GVL_IO.iq_stM2SelectorB.stComOut_EP6002P2/D[2] <-> COM RxPDO-Map Outputs Channel 2/Data Out 2
//     SerialComm Outputs/GVL_IO.iq_stM2SelectorB.stComOut_EP6002P2/D[3] <-> COM RxPDO-Map Outputs Channel 2/Data Out 3
//     SerialComm Outputs/GVL_IO.iq_stM2SelectorB.stComOut_EP6002P2/D[4] <-> COM RxPDO-Map Outputs Channel 2/Data Out 4
//     SerialComm Outputs/GVL_IO.iq_stM2SelectorB.stComOut_EP6002P2/D[5] <-> COM RxPDO-Map Outputs Channel 2/Data Out 5
//     SerialComm Outputs/GVL_IO.iq_stM2SelectorB.stComOut_EP6002P2/D[6] <-> COM RxPDO-Map Outputs Channel 2/Data Out 6
//     SerialComm Outputs/GVL_IO.iq_stM2SelectorB.stComOut_EP6002P2/D[7] <-> COM RxPDO-Map Outputs Channel 2/Data Out 7
//     SerialComm Outputs/GVL_IO.iq_stM2SelectorB.stComOut_EP6002P2/D[8] <-> COM RxPDO-Map Outputs Channel 2/Data Out 8
//     SerialComm Outputs/GVL_IO.iq_stM2SelectorB.stComOut_EP6002P2/D[9] <-> COM RxPDO-Map Outputs Channel 2/Data Out 9
//   SDSM3/SDSM3 Instance <-> MAIN (EtherCAT)/M3 Selector A Digital IO (EP2338-1001)
//     PlcTask Inputs/GVL_IO.iq_stM3SelectorA.i_EP2338_Ch{5..8} <-> Channel {5..8}/Input  (4 links)
//     PlcTask Outputs/GVL_IO.iq_stM3SelectorA.q_EP2338_Ch{1..4} <-> Channel {9..12}/Output  (4 links)
//   SDSM3/SDSM3 Instance <-> MAIN (EtherCAT)/M3 Selector A Mass Flow Meter (Mass Flow / Pressure Controller - Slave)
//     PlcTask Inputs/GVL_IO.iq_stM3SelectorA.i_RawUnit <-> TxPDO/Unit
//     PlcTask Inputs/GVL_IO.iq_stM3SelectorA.i_mfmFlow <-> TxPDO/fMeasure
//   SDSM3/SDSM3 Instance <-> MAIN (EtherCAT)/M3 Selector A Serial IO (EP6002-0002)
//     PlcTask Inputs/GVL_IO.iq_stM3SelectorA.stComIn_EP6002P1/D[0] <-> COM TxPDO-Map Inputs Channel 1/Data In 0
//     PlcTask Inputs/GVL_IO.iq_stM3SelectorA.stComIn_EP6002P1/D[10] <-> COM TxPDO-Map Inputs Channel 1/Data In 10
//     PlcTask Inputs/GVL_IO.iq_stM3SelectorA.stComIn_EP6002P1/D[11] <-> COM TxPDO-Map Inputs Channel 1/Data In 11
//     PlcTask Inputs/GVL_IO.iq_stM3SelectorA.stComIn_EP6002P1/D[12] <-> COM TxPDO-Map Inputs Channel 1/Data In 12
//     PlcTask Inputs/GVL_IO.iq_stM3SelectorA.stComIn_EP6002P1/D[13] <-> COM TxPDO-Map Inputs Channel 1/Data In 13
//     PlcTask Inputs/GVL_IO.iq_stM3SelectorA.stComIn_EP6002P1/D[14] <-> COM TxPDO-Map Inputs Channel 1/Data In 14
//     PlcTask Inputs/GVL_IO.iq_stM3SelectorA.stComIn_EP6002P1/D[15] <-> COM TxPDO-Map Inputs Channel 1/Data In 15
//     PlcTask Inputs/GVL_IO.iq_stM3SelectorA.stComIn_EP6002P1/D[16] <-> COM TxPDO-Map Inputs Channel 1/Data In 16
//     PlcTask Inputs/GVL_IO.iq_stM3SelectorA.stComIn_EP6002P1/D[17] <-> COM TxPDO-Map Inputs Channel 1/Data In 17
//     PlcTask Inputs/GVL_IO.iq_stM3SelectorA.stComIn_EP6002P1/D[18] <-> COM TxPDO-Map Inputs Channel 1/Data In 18
//     PlcTask Inputs/GVL_IO.iq_stM3SelectorA.stComIn_EP6002P1/D[19] <-> COM TxPDO-Map Inputs Channel 1/Data In 19
//     PlcTask Inputs/GVL_IO.iq_stM3SelectorA.stComIn_EP6002P1/D[1] <-> COM TxPDO-Map Inputs Channel 1/Data In 1
//     PlcTask Inputs/GVL_IO.iq_stM3SelectorA.stComIn_EP6002P1/D[20] <-> COM TxPDO-Map Inputs Channel 1/Data In 20
//     PlcTask Inputs/GVL_IO.iq_stM3SelectorA.stComIn_EP6002P1/D[21] <-> COM TxPDO-Map Inputs Channel 1/Data In 21
//     PlcTask Inputs/GVL_IO.iq_stM3SelectorA.stComIn_EP6002P1/D[2] <-> COM TxPDO-Map Inputs Channel 1/Data In 2
//     PlcTask Inputs/GVL_IO.iq_stM3SelectorA.stComIn_EP6002P1/D[3] <-> COM TxPDO-Map Inputs Channel 1/Data In 3
//     PlcTask Inputs/GVL_IO.iq_stM3SelectorA.stComIn_EP6002P1/D[4] <-> COM TxPDO-Map Inputs Channel 1/Data In 4
//     PlcTask Inputs/GVL_IO.iq_stM3SelectorA.stComIn_EP6002P1/D[5] <-> COM TxPDO-Map Inputs Channel 1/Data In 5
//     PlcTask Inputs/GVL_IO.iq_stM3SelectorA.stComIn_EP6002P1/D[6] <-> COM TxPDO-Map Inputs Channel 1/Data In 6
//     PlcTask Inputs/GVL_IO.iq_stM3SelectorA.stComIn_EP6002P1/D[7] <-> COM TxPDO-Map Inputs Channel 1/Data In 7
//     PlcTask Inputs/GVL_IO.iq_stM3SelectorA.stComIn_EP6002P1/D[8] <-> COM TxPDO-Map Inputs Channel 1/Data In 8
//     PlcTask Inputs/GVL_IO.iq_stM3SelectorA.stComIn_EP6002P1/D[9] <-> COM TxPDO-Map Inputs Channel 1/Data In 9
//     PlcTask Inputs/GVL_IO.iq_stM3SelectorA.stComIn_EP6002P2/D[0] <-> COM TxPDO-Map Inputs Channel 2/Data In 0
//     PlcTask Inputs/GVL_IO.iq_stM3SelectorA.stComIn_EP6002P2/D[10] <-> COM TxPDO-Map Inputs Channel 2/Data In 10
//     PlcTask Inputs/GVL_IO.iq_stM3SelectorA.stComIn_EP6002P2/D[11] <-> COM TxPDO-Map Inputs Channel 2/Data In 11
//     PlcTask Inputs/GVL_IO.iq_stM3SelectorA.stComIn_EP6002P2/D[12] <-> COM TxPDO-Map Inputs Channel 2/Data In 12
//     PlcTask Inputs/GVL_IO.iq_stM3SelectorA.stComIn_EP6002P2/D[13] <-> COM TxPDO-Map Inputs Channel 2/Data In 13
//     PlcTask Inputs/GVL_IO.iq_stM3SelectorA.stComIn_EP6002P2/D[14] <-> COM TxPDO-Map Inputs Channel 2/Data In 14
//     PlcTask Inputs/GVL_IO.iq_stM3SelectorA.stComIn_EP6002P2/D[15] <-> COM TxPDO-Map Inputs Channel 2/Data In 15
//     PlcTask Inputs/GVL_IO.iq_stM3SelectorA.stComIn_EP6002P2/D[16] <-> COM TxPDO-Map Inputs Channel 2/Data In 16
//     PlcTask Inputs/GVL_IO.iq_stM3SelectorA.stComIn_EP6002P2/D[17] <-> COM TxPDO-Map Inputs Channel 2/Data In 17
//     PlcTask Inputs/GVL_IO.iq_stM3SelectorA.stComIn_EP6002P2/D[18] <-> COM TxPDO-Map Inputs Channel 2/Data In 18
//     PlcTask Inputs/GVL_IO.iq_stM3SelectorA.stComIn_EP6002P2/D[19] <-> COM TxPDO-Map Inputs Channel 2/Data In 19
//     PlcTask Inputs/GVL_IO.iq_stM3SelectorA.stComIn_EP6002P2/D[1] <-> COM TxPDO-Map Inputs Channel 2/Data In 1
//     PlcTask Inputs/GVL_IO.iq_stM3SelectorA.stComIn_EP6002P2/D[20] <-> COM TxPDO-Map Inputs Channel 2/Data In 20
//     PlcTask Inputs/GVL_IO.iq_stM3SelectorA.stComIn_EP6002P2/D[21] <-> COM TxPDO-Map Inputs Channel 2/Data In 21
//     PlcTask Inputs/GVL_IO.iq_stM3SelectorA.stComIn_EP6002P2/D[2] <-> COM TxPDO-Map Inputs Channel 2/Data In 2
//     PlcTask Inputs/GVL_IO.iq_stM3SelectorA.stComIn_EP6002P2/D[3] <-> COM TxPDO-Map Inputs Channel 2/Data In 3
//     PlcTask Inputs/GVL_IO.iq_stM3SelectorA.stComIn_EP6002P2/D[4] <-> COM TxPDO-Map Inputs Channel 2/Data In 4
//     PlcTask Inputs/GVL_IO.iq_stM3SelectorA.stComIn_EP6002P2/D[5] <-> COM TxPDO-Map Inputs Channel 2/Data In 5
//     PlcTask Inputs/GVL_IO.iq_stM3SelectorA.stComIn_EP6002P2/D[6] <-> COM TxPDO-Map Inputs Channel 2/Data In 6
//     PlcTask Inputs/GVL_IO.iq_stM3SelectorA.stComIn_EP6002P2/D[7] <-> COM TxPDO-Map Inputs Channel 2/Data In 7
//     PlcTask Inputs/GVL_IO.iq_stM3SelectorA.stComIn_EP6002P2/D[8] <-> COM TxPDO-Map Inputs Channel 2/Data In 8
//     PlcTask Inputs/GVL_IO.iq_stM3SelectorA.stComIn_EP6002P2/D[9] <-> COM TxPDO-Map Inputs Channel 2/Data In 9
//     PlcTask Inputs/GVL_IO.iq_stM3SelectorA.stComIn_EP6002P1/Status <-> COM TxPDO-Map Inputs Channel 1/Status
//     PlcTask Inputs/GVL_IO.iq_stM3SelectorA.stComIn_EP6002P2/Status <-> COM TxPDO-Map Inputs Channel 2/Status
//     PlcTask Outputs/GVL_IO.iq_stM3SelectorA.stComOut_EP6002P1/Ctrl <-> COM RxPDO-Map Outputs Channel 1/Ctrl
//     PlcTask Outputs/GVL_IO.iq_stM3SelectorA.stComOut_EP6002P2/Ctrl <-> COM RxPDO-Map Outputs Channel 2/Ctrl
//     PlcTask Outputs/GVL_IO.iq_stM3SelectorA.stComOut_EP6002P1/D[0] <-> COM RxPDO-Map Outputs Channel 1/Data Out 0
//     PlcTask Outputs/GVL_IO.iq_stM3SelectorA.stComOut_EP6002P1/D[10] <-> COM RxPDO-Map Outputs Channel 1/Data Out 10
//     PlcTask Outputs/GVL_IO.iq_stM3SelectorA.stComOut_EP6002P1/D[11] <-> COM RxPDO-Map Outputs Channel 1/Data Out 11
//     PlcTask Outputs/GVL_IO.iq_stM3SelectorA.stComOut_EP6002P1/D[12] <-> COM RxPDO-Map Outputs Channel 1/Data Out 12
//     PlcTask Outputs/GVL_IO.iq_stM3SelectorA.stComOut_EP6002P1/D[13] <-> COM RxPDO-Map Outputs Channel 1/Data Out 13
//     PlcTask Outputs/GVL_IO.iq_stM3SelectorA.stComOut_EP6002P1/D[14] <-> COM RxPDO-Map Outputs Channel 1/Data Out 14
//     PlcTask Outputs/GVL_IO.iq_stM3SelectorA.stComOut_EP6002P1/D[15] <-> COM RxPDO-Map Outputs Channel 1/Data Out 15
//     PlcTask Outputs/GVL_IO.iq_stM3SelectorA.stComOut_EP6002P1/D[16] <-> COM RxPDO-Map Outputs Channel 1/Data Out 16
//     PlcTask Outputs/GVL_IO.iq_stM3SelectorA.stComOut_EP6002P1/D[17] <-> COM RxPDO-Map Outputs Channel 1/Data Out 17
//     PlcTask Outputs/GVL_IO.iq_stM3SelectorA.stComOut_EP6002P1/D[18] <-> COM RxPDO-Map Outputs Channel 1/Data Out 18
//     PlcTask Outputs/GVL_IO.iq_stM3SelectorA.stComOut_EP6002P1/D[19] <-> COM RxPDO-Map Outputs Channel 1/Data Out 19
//     PlcTask Outputs/GVL_IO.iq_stM3SelectorA.stComOut_EP6002P1/D[1] <-> COM RxPDO-Map Outputs Channel 1/Data Out 1
//     PlcTask Outputs/GVL_IO.iq_stM3SelectorA.stComOut_EP6002P1/D[20] <-> COM RxPDO-Map Outputs Channel 1/Data Out 20
//     PlcTask Outputs/GVL_IO.iq_stM3SelectorA.stComOut_EP6002P1/D[21] <-> COM RxPDO-Map Outputs Channel 1/Data Out 21
//     PlcTask Outputs/GVL_IO.iq_stM3SelectorA.stComOut_EP6002P1/D[2] <-> COM RxPDO-Map Outputs Channel 1/Data Out 2
//     PlcTask Outputs/GVL_IO.iq_stM3SelectorA.stComOut_EP6002P1/D[3] <-> COM RxPDO-Map Outputs Channel 1/Data Out 3
//     PlcTask Outputs/GVL_IO.iq_stM3SelectorA.stComOut_EP6002P1/D[4] <-> COM RxPDO-Map Outputs Channel 1/Data Out 4
//     PlcTask Outputs/GVL_IO.iq_stM3SelectorA.stComOut_EP6002P1/D[5] <-> COM RxPDO-Map Outputs Channel 1/Data Out 5
//     PlcTask Outputs/GVL_IO.iq_stM3SelectorA.stComOut_EP6002P1/D[6] <-> COM RxPDO-Map Outputs Channel 1/Data Out 6
//     PlcTask Outputs/GVL_IO.iq_stM3SelectorA.stComOut_EP6002P1/D[7] <-> COM RxPDO-Map Outputs Channel 1/Data Out 7
//     PlcTask Outputs/GVL_IO.iq_stM3SelectorA.stComOut_EP6002P1/D[8] <-> COM RxPDO-Map Outputs Channel 1/Data Out 8
//     PlcTask Outputs/GVL_IO.iq_stM3SelectorA.stComOut_EP6002P1/D[9] <-> COM RxPDO-Map Outputs Channel 1/Data Out 9
//     PlcTask Outputs/GVL_IO.iq_stM3SelectorA.stComOut_EP6002P2/D[0] <-> COM RxPDO-Map Outputs Channel 2/Data Out 0
//     PlcTask Outputs/GVL_IO.iq_stM3SelectorA.stComOut_EP6002P2/D[10] <-> COM RxPDO-Map Outputs Channel 2/Data Out 10
//     PlcTask Outputs/GVL_IO.iq_stM3SelectorA.stComOut_EP6002P2/D[11] <-> COM RxPDO-Map Outputs Channel 2/Data Out 11
//     PlcTask Outputs/GVL_IO.iq_stM3SelectorA.stComOut_EP6002P2/D[12] <-> COM RxPDO-Map Outputs Channel 2/Data Out 12
//     PlcTask Outputs/GVL_IO.iq_stM3SelectorA.stComOut_EP6002P2/D[13] <-> COM RxPDO-Map Outputs Channel 2/Data Out 13
//     PlcTask Outputs/GVL_IO.iq_stM3SelectorA.stComOut_EP6002P2/D[14] <-> COM RxPDO-Map Outputs Channel 2/Data Out 14
//     PlcTask Outputs/GVL_IO.iq_stM3SelectorA.stComOut_EP6002P2/D[15] <-> COM RxPDO-Map Outputs Channel 2/Data Out 15
//     PlcTask Outputs/GVL_IO.iq_stM3SelectorA.stComOut_EP6002P2/D[16] <-> COM RxPDO-Map Outputs Channel 2/Data Out 16
//     PlcTask Outputs/GVL_IO.iq_stM3SelectorA.stComOut_EP6002P2/D[17] <-> COM RxPDO-Map Outputs Channel 2/Data Out 17
//     PlcTask Outputs/GVL_IO.iq_stM3SelectorA.stComOut_EP6002P2/D[18] <-> COM RxPDO-Map Outputs Channel 2/Data Out 18
//     PlcTask Outputs/GVL_IO.iq_stM3SelectorA.stComOut_EP6002P2/D[19] <-> COM RxPDO-Map Outputs Channel 2/Data Out 19
//     PlcTask Outputs/GVL_IO.iq_stM3SelectorA.stComOut_EP6002P2/D[1] <-> COM RxPDO-Map Outputs Channel 2/Data Out 1
//     PlcTask Outputs/GVL_IO.iq_stM3SelectorA.stComOut_EP6002P2/D[20] <-> COM RxPDO-Map Outputs Channel 2/Data Out 20
//     PlcTask Outputs/GVL_IO.iq_stM3SelectorA.stComOut_EP6002P2/D[21] <-> COM RxPDO-Map Outputs Channel 2/Data Out 21
//     PlcTask Outputs/GVL_IO.iq_stM3SelectorA.stComOut_EP6002P2/D[2] <-> COM RxPDO-Map Outputs Channel 2/Data Out 2
//     PlcTask Outputs/GVL_IO.iq_stM3SelectorA.stComOut_EP6002P2/D[3] <-> COM RxPDO-Map Outputs Channel 2/Data Out 3
//     PlcTask Outputs/GVL_IO.iq_stM3SelectorA.stComOut_EP6002P2/D[4] <-> COM RxPDO-Map Outputs Channel 2/Data Out 4
//     PlcTask Outputs/GVL_IO.iq_stM3SelectorA.stComOut_EP6002P2/D[5] <-> COM RxPDO-Map Outputs Channel 2/Data Out 5
//     PlcTask Outputs/GVL_IO.iq_stM3SelectorA.stComOut_EP6002P2/D[6] <-> COM RxPDO-Map Outputs Channel 2/Data Out 6
//     PlcTask Outputs/GVL_IO.iq_stM3SelectorA.stComOut_EP6002P2/D[7] <-> COM RxPDO-Map Outputs Channel 2/Data Out 7
//     PlcTask Outputs/GVL_IO.iq_stM3SelectorA.stComOut_EP6002P2/D[8] <-> COM RxPDO-Map Outputs Channel 2/Data Out 8
//     PlcTask Outputs/GVL_IO.iq_stM3SelectorA.stComOut_EP6002P2/D[9] <-> COM RxPDO-Map Outputs Channel 2/Data Out 9
//   SDSM3/SDSM3 Instance <-> MAIN (EtherCAT)/M3 Selector B Digital IO (EP2338-1001)
//     PlcTask Inputs/GVL_IO.iq_stM3SelectorB.i_EP2338_Ch{5..8} <-> Channel {5..8}/Input  (4 links)
//     PlcTask Outputs/GVL_IO.iq_stM3SelectorB.q_EP2338_Ch{1..4} <-> Channel {9..12}/Output  (4 links)
//   SDSM3/SDSM3 Instance <-> MAIN (EtherCAT)/M3 Selector B Mass Flow Meter (Mass Flow / Pressure Controller - Slave)
//     PlcTask Inputs/GVL_IO.iq_stM3SelectorB.i_RawUnit <-> TxPDO/Unit
//     PlcTask Inputs/GVL_IO.iq_stM3SelectorB.i_mfmFlow <-> TxPDO/fMeasure
//   SDSM3/SDSM3 Instance <-> MAIN (EtherCAT)/M3 Selector B Serial IO (EP6002-0002)
//     PlcTask Inputs/GVL_IO.iq_stM3SelectorB.stComIn_EP6002P1/D[0] <-> COM TxPDO-Map Inputs Channel 1/Data In 0
//     PlcTask Inputs/GVL_IO.iq_stM3SelectorB.stComIn_EP6002P1/D[10] <-> COM TxPDO-Map Inputs Channel 1/Data In 10
//     PlcTask Inputs/GVL_IO.iq_stM3SelectorB.stComIn_EP6002P1/D[11] <-> COM TxPDO-Map Inputs Channel 1/Data In 11
//     PlcTask Inputs/GVL_IO.iq_stM3SelectorB.stComIn_EP6002P1/D[12] <-> COM TxPDO-Map Inputs Channel 1/Data In 12
//     PlcTask Inputs/GVL_IO.iq_stM3SelectorB.stComIn_EP6002P1/D[13] <-> COM TxPDO-Map Inputs Channel 1/Data In 13
//     PlcTask Inputs/GVL_IO.iq_stM3SelectorB.stComIn_EP6002P1/D[14] <-> COM TxPDO-Map Inputs Channel 1/Data In 14
//     PlcTask Inputs/GVL_IO.iq_stM3SelectorB.stComIn_EP6002P1/D[15] <-> COM TxPDO-Map Inputs Channel 1/Data In 15
//     PlcTask Inputs/GVL_IO.iq_stM3SelectorB.stComIn_EP6002P1/D[16] <-> COM TxPDO-Map Inputs Channel 1/Data In 16
//     PlcTask Inputs/GVL_IO.iq_stM3SelectorB.stComIn_EP6002P1/D[17] <-> COM TxPDO-Map Inputs Channel 1/Data In 17
//     PlcTask Inputs/GVL_IO.iq_stM3SelectorB.stComIn_EP6002P1/D[18] <-> COM TxPDO-Map Inputs Channel 1/Data In 18
//     PlcTask Inputs/GVL_IO.iq_stM3SelectorB.stComIn_EP6002P1/D[19] <-> COM TxPDO-Map Inputs Channel 1/Data In 19
//     PlcTask Inputs/GVL_IO.iq_stM3SelectorB.stComIn_EP6002P1/D[1] <-> COM TxPDO-Map Inputs Channel 1/Data In 1
//     PlcTask Inputs/GVL_IO.iq_stM3SelectorB.stComIn_EP6002P1/D[20] <-> COM TxPDO-Map Inputs Channel 1/Data In 20
//     PlcTask Inputs/GVL_IO.iq_stM3SelectorB.stComIn_EP6002P1/D[21] <-> COM TxPDO-Map Inputs Channel 1/Data In 21
//     PlcTask Inputs/GVL_IO.iq_stM3SelectorB.stComIn_EP6002P1/D[2] <-> COM TxPDO-Map Inputs Channel 1/Data In 2
//     PlcTask Inputs/GVL_IO.iq_stM3SelectorB.stComIn_EP6002P1/D[3] <-> COM TxPDO-Map Inputs Channel 1/Data In 3
//     PlcTask Inputs/GVL_IO.iq_stM3SelectorB.stComIn_EP6002P1/D[4] <-> COM TxPDO-Map Inputs Channel 1/Data In 4
//     PlcTask Inputs/GVL_IO.iq_stM3SelectorB.stComIn_EP6002P1/D[5] <-> COM TxPDO-Map Inputs Channel 1/Data In 5
//     PlcTask Inputs/GVL_IO.iq_stM3SelectorB.stComIn_EP6002P1/D[6] <-> COM TxPDO-Map Inputs Channel 1/Data In 6
//     PlcTask Inputs/GVL_IO.iq_stM3SelectorB.stComIn_EP6002P1/D[7] <-> COM TxPDO-Map Inputs Channel 1/Data In 7
//     PlcTask Inputs/GVL_IO.iq_stM3SelectorB.stComIn_EP6002P1/D[8] <-> COM TxPDO-Map Inputs Channel 1/Data In 8
//     PlcTask Inputs/GVL_IO.iq_stM3SelectorB.stComIn_EP6002P1/D[9] <-> COM TxPDO-Map Inputs Channel 1/Data In 9
//     PlcTask Inputs/GVL_IO.iq_stM3SelectorB.stComIn_EP6002P2/D[0] <-> COM TxPDO-Map Inputs Channel 2/Data In 0
//     PlcTask Inputs/GVL_IO.iq_stM3SelectorB.stComIn_EP6002P2/D[10] <-> COM TxPDO-Map Inputs Channel 2/Data In 10
//     PlcTask Inputs/GVL_IO.iq_stM3SelectorB.stComIn_EP6002P2/D[11] <-> COM TxPDO-Map Inputs Channel 2/Data In 11
//     PlcTask Inputs/GVL_IO.iq_stM3SelectorB.stComIn_EP6002P2/D[12] <-> COM TxPDO-Map Inputs Channel 2/Data In 12
//     PlcTask Inputs/GVL_IO.iq_stM3SelectorB.stComIn_EP6002P2/D[13] <-> COM TxPDO-Map Inputs Channel 2/Data In 13
//     PlcTask Inputs/GVL_IO.iq_stM3SelectorB.stComIn_EP6002P2/D[14] <-> COM TxPDO-Map Inputs Channel 2/Data In 14
//     PlcTask Inputs/GVL_IO.iq_stM3SelectorB.stComIn_EP6002P2/D[15] <-> COM TxPDO-Map Inputs Channel 2/Data In 15
//     PlcTask Inputs/GVL_IO.iq_stM3SelectorB.stComIn_EP6002P2/D[16] <-> COM TxPDO-Map Inputs Channel 2/Data In 16
//     PlcTask Inputs/GVL_IO.iq_stM3SelectorB.stComIn_EP6002P2/D[17] <-> COM TxPDO-Map Inputs Channel 2/Data In 17
//     PlcTask Inputs/GVL_IO.iq_stM3SelectorB.stComIn_EP6002P2/D[18] <-> COM TxPDO-Map Inputs Channel 2/Data In 18
//     PlcTask Inputs/GVL_IO.iq_stM3SelectorB.stComIn_EP6002P2/D[19] <-> COM TxPDO-Map Inputs Channel 2/Data In 19
//     PlcTask Inputs/GVL_IO.iq_stM3SelectorB.stComIn_EP6002P2/D[1] <-> COM TxPDO-Map Inputs Channel 2/Data In 1
//     PlcTask Inputs/GVL_IO.iq_stM3SelectorB.stComIn_EP6002P2/D[20] <-> COM TxPDO-Map Inputs Channel 2/Data In 20
//     PlcTask Inputs/GVL_IO.iq_stM3SelectorB.stComIn_EP6002P2/D[21] <-> COM TxPDO-Map Inputs Channel 2/Data In 21
//     PlcTask Inputs/GVL_IO.iq_stM3SelectorB.stComIn_EP6002P2/D[2] <-> COM TxPDO-Map Inputs Channel 2/Data In 2
//     PlcTask Inputs/GVL_IO.iq_stM3SelectorB.stComIn_EP6002P2/D[3] <-> COM TxPDO-Map Inputs Channel 2/Data In 3
//     PlcTask Inputs/GVL_IO.iq_stM3SelectorB.stComIn_EP6002P2/D[4] <-> COM TxPDO-Map Inputs Channel 2/Data In 4
//     PlcTask Inputs/GVL_IO.iq_stM3SelectorB.stComIn_EP6002P2/D[5] <-> COM TxPDO-Map Inputs Channel 2/Data In 5
//     PlcTask Inputs/GVL_IO.iq_stM3SelectorB.stComIn_EP6002P2/D[6] <-> COM TxPDO-Map Inputs Channel 2/Data In 6
//     PlcTask Inputs/GVL_IO.iq_stM3SelectorB.stComIn_EP6002P2/D[7] <-> COM TxPDO-Map Inputs Channel 2/Data In 7
//     PlcTask Inputs/GVL_IO.iq_stM3SelectorB.stComIn_EP6002P2/D[8] <-> COM TxPDO-Map Inputs Channel 2/Data In 8
//     PlcTask Inputs/GVL_IO.iq_stM3SelectorB.stComIn_EP6002P2/D[9] <-> COM TxPDO-Map Inputs Channel 2/Data In 9
//     PlcTask Inputs/GVL_IO.iq_stM3SelectorB.stComIn_EP6002P1/Status <-> COM TxPDO-Map Inputs Channel 1/Status
//     PlcTask Inputs/GVL_IO.iq_stM3SelectorB.stComIn_EP6002P2/Status <-> COM TxPDO-Map Inputs Channel 2/Status
//     PlcTask Outputs/GVL_IO.iq_stM3SelectorB.stComOut_EP6002P1/Ctrl <-> COM RxPDO-Map Outputs Channel 1/Ctrl
//     PlcTask Outputs/GVL_IO.iq_stM3SelectorB.stComOut_EP6002P2/Ctrl <-> COM RxPDO-Map Outputs Channel 2/Ctrl
//     PlcTask Outputs/GVL_IO.iq_stM3SelectorB.stComOut_EP6002P1/D[0] <-> COM RxPDO-Map Outputs Channel 1/Data Out 0
//     PlcTask Outputs/GVL_IO.iq_stM3SelectorB.stComOut_EP6002P1/D[10] <-> COM RxPDO-Map Outputs Channel 1/Data Out 10
//     PlcTask Outputs/GVL_IO.iq_stM3SelectorB.stComOut_EP6002P1/D[11] <-> COM RxPDO-Map Outputs Channel 1/Data Out 11
//     PlcTask Outputs/GVL_IO.iq_stM3SelectorB.stComOut_EP6002P1/D[12] <-> COM RxPDO-Map Outputs Channel 1/Data Out 12
//     PlcTask Outputs/GVL_IO.iq_stM3SelectorB.stComOut_EP6002P1/D[13] <-> COM RxPDO-Map Outputs Channel 1/Data Out 13
//     PlcTask Outputs/GVL_IO.iq_stM3SelectorB.stComOut_EP6002P1/D[14] <-> COM RxPDO-Map Outputs Channel 1/Data Out 14
//     PlcTask Outputs/GVL_IO.iq_stM3SelectorB.stComOut_EP6002P1/D[15] <-> COM RxPDO-Map Outputs Channel 1/Data Out 15
//     PlcTask Outputs/GVL_IO.iq_stM3SelectorB.stComOut_EP6002P1/D[16] <-> COM RxPDO-Map Outputs Channel 1/Data Out 16
//     PlcTask Outputs/GVL_IO.iq_stM3SelectorB.stComOut_EP6002P1/D[17] <-> COM RxPDO-Map Outputs Channel 1/Data Out 17
//     PlcTask Outputs/GVL_IO.iq_stM3SelectorB.stComOut_EP6002P1/D[18] <-> COM RxPDO-Map Outputs Channel 1/Data Out 18
//     PlcTask Outputs/GVL_IO.iq_stM3SelectorB.stComOut_EP6002P1/D[19] <-> COM RxPDO-Map Outputs Channel 1/Data Out 19
//     PlcTask Outputs/GVL_IO.iq_stM3SelectorB.stComOut_EP6002P1/D[1] <-> COM RxPDO-Map Outputs Channel 1/Data Out 1
//     PlcTask Outputs/GVL_IO.iq_stM3SelectorB.stComOut_EP6002P1/D[20] <-> COM RxPDO-Map Outputs Channel 1/Data Out 20
//     PlcTask Outputs/GVL_IO.iq_stM3SelectorB.stComOut_EP6002P1/D[21] <-> COM RxPDO-Map Outputs Channel 1/Data Out 21
//     PlcTask Outputs/GVL_IO.iq_stM3SelectorB.stComOut_EP6002P1/D[2] <-> COM RxPDO-Map Outputs Channel 1/Data Out 2
//     PlcTask Outputs/GVL_IO.iq_stM3SelectorB.stComOut_EP6002P1/D[3] <-> COM RxPDO-Map Outputs Channel 1/Data Out 3
//     PlcTask Outputs/GVL_IO.iq_stM3SelectorB.stComOut_EP6002P1/D[4] <-> COM RxPDO-Map Outputs Channel 1/Data Out 4
//     PlcTask Outputs/GVL_IO.iq_stM3SelectorB.stComOut_EP6002P1/D[5] <-> COM RxPDO-Map Outputs Channel 1/Data Out 5
//     PlcTask Outputs/GVL_IO.iq_stM3SelectorB.stComOut_EP6002P1/D[6] <-> COM RxPDO-Map Outputs Channel 1/Data Out 6
//     PlcTask Outputs/GVL_IO.iq_stM3SelectorB.stComOut_EP6002P1/D[7] <-> COM RxPDO-Map Outputs Channel 1/Data Out 7
//     PlcTask Outputs/GVL_IO.iq_stM3SelectorB.stComOut_EP6002P1/D[8] <-> COM RxPDO-Map Outputs Channel 1/Data Out 8
//     PlcTask Outputs/GVL_IO.iq_stM3SelectorB.stComOut_EP6002P1/D[9] <-> COM RxPDO-Map Outputs Channel 1/Data Out 9
//     PlcTask Outputs/GVL_IO.iq_stM3SelectorB.stComOut_EP6002P2/D[0] <-> COM RxPDO-Map Outputs Channel 2/Data Out 0
//     PlcTask Outputs/GVL_IO.iq_stM3SelectorB.stComOut_EP6002P2/D[10] <-> COM RxPDO-Map Outputs Channel 2/Data Out 10
//     PlcTask Outputs/GVL_IO.iq_stM3SelectorB.stComOut_EP6002P2/D[11] <-> COM RxPDO-Map Outputs Channel 2/Data Out 11
//     PlcTask Outputs/GVL_IO.iq_stM3SelectorB.stComOut_EP6002P2/D[12] <-> COM RxPDO-Map Outputs Channel 2/Data Out 12
//     PlcTask Outputs/GVL_IO.iq_stM3SelectorB.stComOut_EP6002P2/D[13] <-> COM RxPDO-Map Outputs Channel 2/Data Out 13
//     PlcTask Outputs/GVL_IO.iq_stM3SelectorB.stComOut_EP6002P2/D[14] <-> COM RxPDO-Map Outputs Channel 2/Data Out 14
//     PlcTask Outputs/GVL_IO.iq_stM3SelectorB.stComOut_EP6002P2/D[15] <-> COM RxPDO-Map Outputs Channel 2/Data Out 15
//     PlcTask Outputs/GVL_IO.iq_stM3SelectorB.stComOut_EP6002P2/D[16] <-> COM RxPDO-Map Outputs Channel 2/Data Out 16
//     PlcTask Outputs/GVL_IO.iq_stM3SelectorB.stComOut_EP6002P2/D[17] <-> COM RxPDO-Map Outputs Channel 2/Data Out 17
//     PlcTask Outputs/GVL_IO.iq_stM3SelectorB.stComOut_EP6002P2/D[18] <-> COM RxPDO-Map Outputs Channel 2/Data Out 18
//     PlcTask Outputs/GVL_IO.iq_stM3SelectorB.stComOut_EP6002P2/D[19] <-> COM RxPDO-Map Outputs Channel 2/Data Out 19
//     PlcTask Outputs/GVL_IO.iq_stM3SelectorB.stComOut_EP6002P2/D[1] <-> COM RxPDO-Map Outputs Channel 2/Data Out 1
//     PlcTask Outputs/GVL_IO.iq_stM3SelectorB.stComOut_EP6002P2/D[20] <-> COM RxPDO-Map Outputs Channel 2/Data Out 20
//     PlcTask Outputs/GVL_IO.iq_stM3SelectorB.stComOut_EP6002P2/D[21] <-> COM RxPDO-Map Outputs Channel 2/Data Out 21
//     PlcTask Outputs/GVL_IO.iq_stM3SelectorB.stComOut_EP6002P2/D[2] <-> COM RxPDO-Map Outputs Channel 2/Data Out 2
//     PlcTask Outputs/GVL_IO.iq_stM3SelectorB.stComOut_EP6002P2/D[3] <-> COM RxPDO-Map Outputs Channel 2/Data Out 3
//     PlcTask Outputs/GVL_IO.iq_stM3SelectorB.stComOut_EP6002P2/D[4] <-> COM RxPDO-Map Outputs Channel 2/Data Out 4
//     PlcTask Outputs/GVL_IO.iq_stM3SelectorB.stComOut_EP6002P2/D[5] <-> COM RxPDO-Map Outputs Channel 2/Data Out 5
//     PlcTask Outputs/GVL_IO.iq_stM3SelectorB.stComOut_EP6002P2/D[6] <-> COM RxPDO-Map Outputs Channel 2/Data Out 6
//     PlcTask Outputs/GVL_IO.iq_stM3SelectorB.stComOut_EP6002P2/D[7] <-> COM RxPDO-Map Outputs Channel 2/Data Out 7
//     PlcTask Outputs/GVL_IO.iq_stM3SelectorB.stComOut_EP6002P2/D[8] <-> COM RxPDO-Map Outputs Channel 2/Data Out 8
//     PlcTask Outputs/GVL_IO.iq_stM3SelectorB.stComOut_EP6002P2/D[9] <-> COM RxPDO-Map Outputs Channel 2/Data Out 9
//   SDSM3/SDSM3 Instance <-> MAIN (EtherCAT)/PCM A (EP3174-0002)
//     PlcTask Inputs/GVL_IO.iq_stPressCtrlA.i_EP3174_Ch{1..4} <-> AI Standard Channel {1..4}/Value  (4 links)
//   SDSM3/SDSM3 Instance <-> MAIN (EtherCAT)/PCM A (EP4374-0002)
//     PlcTask Inputs/GVL_IO.iq_stPressCtrlA.i_EP4374_Ch1 <-> AI Inputs Channel 1/Value
//     PlcTask Inputs/GVL_IO.iq_stPressCtrlA.i_EP4374_Ch2 <-> AI Inputs Channel 2/Value
//     PlcTask Outputs/GVL_IO.iq_stPressCtrlA.q_EP4374_Ch3 <-> AO Outputs Channel 3/Analog output
//     PlcTask Outputs/GVL_IO.iq_stPressCtrlA.q_EP4374_Ch4 <-> AO Outputs Channel 4/Analog output
//   SDSM3/SDSM3 Instance <-> MAIN (EtherCAT)/PCM A (EP6002-0002)
//     PlcTask Inputs/GVL_IO.iq_stPressCtrlA.stComIn_EP6002P1/D[0] <-> COM TxPDO-Map Inputs Channel 1/Data In 0
//     PlcTask Inputs/GVL_IO.iq_stPressCtrlA.stComIn_EP6002P1/D[10] <-> COM TxPDO-Map Inputs Channel 1/Data In 10
//     PlcTask Inputs/GVL_IO.iq_stPressCtrlA.stComIn_EP6002P1/D[11] <-> COM TxPDO-Map Inputs Channel 1/Data In 11
//     PlcTask Inputs/GVL_IO.iq_stPressCtrlA.stComIn_EP6002P1/D[12] <-> COM TxPDO-Map Inputs Channel 1/Data In 12
//     PlcTask Inputs/GVL_IO.iq_stPressCtrlA.stComIn_EP6002P1/D[13] <-> COM TxPDO-Map Inputs Channel 1/Data In 13
//     PlcTask Inputs/GVL_IO.iq_stPressCtrlA.stComIn_EP6002P1/D[14] <-> COM TxPDO-Map Inputs Channel 1/Data In 14
//     PlcTask Inputs/GVL_IO.iq_stPressCtrlA.stComIn_EP6002P1/D[15] <-> COM TxPDO-Map Inputs Channel 1/Data In 15
//     PlcTask Inputs/GVL_IO.iq_stPressCtrlA.stComIn_EP6002P1/D[16] <-> COM TxPDO-Map Inputs Channel 1/Data In 16
//     PlcTask Inputs/GVL_IO.iq_stPressCtrlA.stComIn_EP6002P1/D[17] <-> COM TxPDO-Map Inputs Channel 1/Data In 17
//     PlcTask Inputs/GVL_IO.iq_stPressCtrlA.stComIn_EP6002P1/D[18] <-> COM TxPDO-Map Inputs Channel 1/Data In 18
//     PlcTask Inputs/GVL_IO.iq_stPressCtrlA.stComIn_EP6002P1/D[19] <-> COM TxPDO-Map Inputs Channel 1/Data In 19
//     PlcTask Inputs/GVL_IO.iq_stPressCtrlA.stComIn_EP6002P1/D[1] <-> COM TxPDO-Map Inputs Channel 1/Data In 1
//     PlcTask Inputs/GVL_IO.iq_stPressCtrlA.stComIn_EP6002P1/D[20] <-> COM TxPDO-Map Inputs Channel 1/Data In 20
//     PlcTask Inputs/GVL_IO.iq_stPressCtrlA.stComIn_EP6002P1/D[21] <-> COM TxPDO-Map Inputs Channel 1/Data In 21
//     PlcTask Inputs/GVL_IO.iq_stPressCtrlA.stComIn_EP6002P1/D[2] <-> COM TxPDO-Map Inputs Channel 1/Data In 2
//     PlcTask Inputs/GVL_IO.iq_stPressCtrlA.stComIn_EP6002P1/D[3] <-> COM TxPDO-Map Inputs Channel 1/Data In 3
//     PlcTask Inputs/GVL_IO.iq_stPressCtrlA.stComIn_EP6002P1/D[4] <-> COM TxPDO-Map Inputs Channel 1/Data In 4
//     PlcTask Inputs/GVL_IO.iq_stPressCtrlA.stComIn_EP6002P1/D[5] <-> COM TxPDO-Map Inputs Channel 1/Data In 5
//     PlcTask Inputs/GVL_IO.iq_stPressCtrlA.stComIn_EP6002P1/D[6] <-> COM TxPDO-Map Inputs Channel 1/Data In 6
//     PlcTask Inputs/GVL_IO.iq_stPressCtrlA.stComIn_EP6002P1/D[7] <-> COM TxPDO-Map Inputs Channel 1/Data In 7
//     PlcTask Inputs/GVL_IO.iq_stPressCtrlA.stComIn_EP6002P1/D[8] <-> COM TxPDO-Map Inputs Channel 1/Data In 8
//     PlcTask Inputs/GVL_IO.iq_stPressCtrlA.stComIn_EP6002P1/D[9] <-> COM TxPDO-Map Inputs Channel 1/Data In 9
//     PlcTask Inputs/GVL_IO.iq_stPressCtrlA.stComIn_EP6002P2/D[0] <-> COM TxPDO-Map Inputs Channel 2/Data In 0
//     PlcTask Inputs/GVL_IO.iq_stPressCtrlA.stComIn_EP6002P2/D[10] <-> COM TxPDO-Map Inputs Channel 2/Data In 10
//     PlcTask Inputs/GVL_IO.iq_stPressCtrlA.stComIn_EP6002P2/D[11] <-> COM TxPDO-Map Inputs Channel 2/Data In 11
//     PlcTask Inputs/GVL_IO.iq_stPressCtrlA.stComIn_EP6002P2/D[12] <-> COM TxPDO-Map Inputs Channel 2/Data In 12
//     PlcTask Inputs/GVL_IO.iq_stPressCtrlA.stComIn_EP6002P2/D[13] <-> COM TxPDO-Map Inputs Channel 2/Data In 13
//     PlcTask Inputs/GVL_IO.iq_stPressCtrlA.stComIn_EP6002P2/D[14] <-> COM TxPDO-Map Inputs Channel 2/Data In 14
//     PlcTask Inputs/GVL_IO.iq_stPressCtrlA.stComIn_EP6002P2/D[15] <-> COM TxPDO-Map Inputs Channel 2/Data In 15
//     PlcTask Inputs/GVL_IO.iq_stPressCtrlA.stComIn_EP6002P2/D[16] <-> COM TxPDO-Map Inputs Channel 2/Data In 16
//     PlcTask Inputs/GVL_IO.iq_stPressCtrlA.stComIn_EP6002P2/D[17] <-> COM TxPDO-Map Inputs Channel 2/Data In 17
//     PlcTask Inputs/GVL_IO.iq_stPressCtrlA.stComIn_EP6002P2/D[18] <-> COM TxPDO-Map Inputs Channel 2/Data In 18
//     PlcTask Inputs/GVL_IO.iq_stPressCtrlA.stComIn_EP6002P2/D[19] <-> COM TxPDO-Map Inputs Channel 2/Data In 19
//     PlcTask Inputs/GVL_IO.iq_stPressCtrlA.stComIn_EP6002P2/D[1] <-> COM TxPDO-Map Inputs Channel 2/Data In 1
//     PlcTask Inputs/GVL_IO.iq_stPressCtrlA.stComIn_EP6002P2/D[20] <-> COM TxPDO-Map Inputs Channel 2/Data In 20
//     PlcTask Inputs/GVL_IO.iq_stPressCtrlA.stComIn_EP6002P2/D[21] <-> COM TxPDO-Map Inputs Channel 2/Data In 21
//     PlcTask Inputs/GVL_IO.iq_stPressCtrlA.stComIn_EP6002P2/D[2] <-> COM TxPDO-Map Inputs Channel 2/Data In 2
//     PlcTask Inputs/GVL_IO.iq_stPressCtrlA.stComIn_EP6002P2/D[3] <-> COM TxPDO-Map Inputs Channel 2/Data In 3
//     PlcTask Inputs/GVL_IO.iq_stPressCtrlA.stComIn_EP6002P2/D[4] <-> COM TxPDO-Map Inputs Channel 2/Data In 4
//     PlcTask Inputs/GVL_IO.iq_stPressCtrlA.stComIn_EP6002P2/D[5] <-> COM TxPDO-Map Inputs Channel 2/Data In 5
//     PlcTask Inputs/GVL_IO.iq_stPressCtrlA.stComIn_EP6002P2/D[6] <-> COM TxPDO-Map Inputs Channel 2/Data In 6
//     PlcTask Inputs/GVL_IO.iq_stPressCtrlA.stComIn_EP6002P2/D[7] <-> COM TxPDO-Map Inputs Channel 2/Data In 7
//     PlcTask Inputs/GVL_IO.iq_stPressCtrlA.stComIn_EP6002P2/D[8] <-> COM TxPDO-Map Inputs Channel 2/Data In 8
//     PlcTask Inputs/GVL_IO.iq_stPressCtrlA.stComIn_EP6002P2/D[9] <-> COM TxPDO-Map Inputs Channel 2/Data In 9
//     PlcTask Inputs/GVL_IO.iq_stPressCtrlA.stComIn_EP6002P1/Status <-> COM TxPDO-Map Inputs Channel 1/Status
//     PlcTask Inputs/GVL_IO.iq_stPressCtrlA.stComIn_EP6002P2/Status <-> COM TxPDO-Map Inputs Channel 2/Status
//     PlcTask Outputs/GVL_IO.iq_stPressCtrlA.stComOut_EP6002P1/Ctrl <-> COM RxPDO-Map Outputs Channel 1/Ctrl
//     PlcTask Outputs/GVL_IO.iq_stPressCtrlA.stComOut_EP6002P2/Ctrl <-> COM RxPDO-Map Outputs Channel 2/Ctrl
//     PlcTask Outputs/GVL_IO.iq_stPressCtrlA.stComOut_EP6002P1/D[0] <-> COM RxPDO-Map Outputs Channel 1/Data Out 0
//     PlcTask Outputs/GVL_IO.iq_stPressCtrlA.stComOut_EP6002P1/D[10] <-> COM RxPDO-Map Outputs Channel 1/Data Out 10
//     PlcTask Outputs/GVL_IO.iq_stPressCtrlA.stComOut_EP6002P1/D[11] <-> COM RxPDO-Map Outputs Channel 1/Data Out 11
//     PlcTask Outputs/GVL_IO.iq_stPressCtrlA.stComOut_EP6002P1/D[12] <-> COM RxPDO-Map Outputs Channel 1/Data Out 12
//     PlcTask Outputs/GVL_IO.iq_stPressCtrlA.stComOut_EP6002P1/D[13] <-> COM RxPDO-Map Outputs Channel 1/Data Out 13
//     PlcTask Outputs/GVL_IO.iq_stPressCtrlA.stComOut_EP6002P1/D[14] <-> COM RxPDO-Map Outputs Channel 1/Data Out 14
//     PlcTask Outputs/GVL_IO.iq_stPressCtrlA.stComOut_EP6002P1/D[15] <-> COM RxPDO-Map Outputs Channel 1/Data Out 15
//     PlcTask Outputs/GVL_IO.iq_stPressCtrlA.stComOut_EP6002P1/D[16] <-> COM RxPDO-Map Outputs Channel 1/Data Out 16
//     PlcTask Outputs/GVL_IO.iq_stPressCtrlA.stComOut_EP6002P1/D[17] <-> COM RxPDO-Map Outputs Channel 1/Data Out 17
//     PlcTask Outputs/GVL_IO.iq_stPressCtrlA.stComOut_EP6002P1/D[18] <-> COM RxPDO-Map Outputs Channel 1/Data Out 18
//     PlcTask Outputs/GVL_IO.iq_stPressCtrlA.stComOut_EP6002P1/D[19] <-> COM RxPDO-Map Outputs Channel 1/Data Out 19
//     PlcTask Outputs/GVL_IO.iq_stPressCtrlA.stComOut_EP6002P1/D[1] <-> COM RxPDO-Map Outputs Channel 1/Data Out 1
//     PlcTask Outputs/GVL_IO.iq_stPressCtrlA.stComOut_EP6002P1/D[20] <-> COM RxPDO-Map Outputs Channel 1/Data Out 20
//     PlcTask Outputs/GVL_IO.iq_stPressCtrlA.stComOut_EP6002P1/D[21] <-> COM RxPDO-Map Outputs Channel 1/Data Out 21
//     PlcTask Outputs/GVL_IO.iq_stPressCtrlA.stComOut_EP6002P1/D[2] <-> COM RxPDO-Map Outputs Channel 1/Data Out 2
//     PlcTask Outputs/GVL_IO.iq_stPressCtrlA.stComOut_EP6002P1/D[3] <-> COM RxPDO-Map Outputs Channel 1/Data Out 3
//     PlcTask Outputs/GVL_IO.iq_stPressCtrlA.stComOut_EP6002P1/D[4] <-> COM RxPDO-Map Outputs Channel 1/Data Out 4
//     PlcTask Outputs/GVL_IO.iq_stPressCtrlA.stComOut_EP6002P1/D[5] <-> COM RxPDO-Map Outputs Channel 1/Data Out 5
//     PlcTask Outputs/GVL_IO.iq_stPressCtrlA.stComOut_EP6002P1/D[6] <-> COM RxPDO-Map Outputs Channel 1/Data Out 6
//     PlcTask Outputs/GVL_IO.iq_stPressCtrlA.stComOut_EP6002P1/D[7] <-> COM RxPDO-Map Outputs Channel 1/Data Out 7
//     PlcTask Outputs/GVL_IO.iq_stPressCtrlA.stComOut_EP6002P1/D[8] <-> COM RxPDO-Map Outputs Channel 1/Data Out 8
//     PlcTask Outputs/GVL_IO.iq_stPressCtrlA.stComOut_EP6002P1/D[9] <-> COM RxPDO-Map Outputs Channel 1/Data Out 9
//     PlcTask Outputs/GVL_IO.iq_stPressCtrlA.stComOut_EP6002P2/D[0] <-> COM RxPDO-Map Outputs Channel 2/Data Out 0
//     PlcTask Outputs/GVL_IO.iq_stPressCtrlA.stComOut_EP6002P2/D[10] <-> COM RxPDO-Map Outputs Channel 2/Data Out 10
//     PlcTask Outputs/GVL_IO.iq_stPressCtrlA.stComOut_EP6002P2/D[11] <-> COM RxPDO-Map Outputs Channel 2/Data Out 11
//     PlcTask Outputs/GVL_IO.iq_stPressCtrlA.stComOut_EP6002P2/D[12] <-> COM RxPDO-Map Outputs Channel 2/Data Out 12
//     PlcTask Outputs/GVL_IO.iq_stPressCtrlA.stComOut_EP6002P2/D[13] <-> COM RxPDO-Map Outputs Channel 2/Data Out 13
//     PlcTask Outputs/GVL_IO.iq_stPressCtrlA.stComOut_EP6002P2/D[14] <-> COM RxPDO-Map Outputs Channel 2/Data Out 14
//     PlcTask Outputs/GVL_IO.iq_stPressCtrlA.stComOut_EP6002P2/D[15] <-> COM RxPDO-Map Outputs Channel 2/Data Out 15
//     PlcTask Outputs/GVL_IO.iq_stPressCtrlA.stComOut_EP6002P2/D[16] <-> COM RxPDO-Map Outputs Channel 2/Data Out 16
//     PlcTask Outputs/GVL_IO.iq_stPressCtrlA.stComOut_EP6002P2/D[17] <-> COM RxPDO-Map Outputs Channel 2/Data Out 17
//     PlcTask Outputs/GVL_IO.iq_stPressCtrlA.stComOut_EP6002P2/D[18] <-> COM RxPDO-Map Outputs Channel 2/Data Out 18
//     PlcTask Outputs/GVL_IO.iq_stPressCtrlA.stComOut_EP6002P2/D[19] <-> COM RxPDO-Map Outputs Channel 2/Data Out 19
//     PlcTask Outputs/GVL_IO.iq_stPressCtrlA.stComOut_EP6002P2/D[1] <-> COM RxPDO-Map Outputs Channel 2/Data Out 1
//     PlcTask Outputs/GVL_IO.iq_stPressCtrlA.stComOut_EP6002P2/D[20] <-> COM RxPDO-Map Outputs Channel 2/Data Out 20
//     PlcTask Outputs/GVL_IO.iq_stPressCtrlA.stComOut_EP6002P2/D[21] <-> COM RxPDO-Map Outputs Channel 2/Data Out 21
//     PlcTask Outputs/GVL_IO.iq_stPressCtrlA.stComOut_EP6002P2/D[2] <-> COM RxPDO-Map Outputs Channel 2/Data Out 2
//     PlcTask Outputs/GVL_IO.iq_stPressCtrlA.stComOut_EP6002P2/D[3] <-> COM RxPDO-Map Outputs Channel 2/Data Out 3
//     PlcTask Outputs/GVL_IO.iq_stPressCtrlA.stComOut_EP6002P2/D[4] <-> COM RxPDO-Map Outputs Channel 2/Data Out 4
//     PlcTask Outputs/GVL_IO.iq_stPressCtrlA.stComOut_EP6002P2/D[5] <-> COM RxPDO-Map Outputs Channel 2/Data Out 5
//     PlcTask Outputs/GVL_IO.iq_stPressCtrlA.stComOut_EP6002P2/D[6] <-> COM RxPDO-Map Outputs Channel 2/Data Out 6
//     PlcTask Outputs/GVL_IO.iq_stPressCtrlA.stComOut_EP6002P2/D[7] <-> COM RxPDO-Map Outputs Channel 2/Data Out 7
//     PlcTask Outputs/GVL_IO.iq_stPressCtrlA.stComOut_EP6002P2/D[8] <-> COM RxPDO-Map Outputs Channel 2/Data Out 8
//     PlcTask Outputs/GVL_IO.iq_stPressCtrlA.stComOut_EP6002P2/D[9] <-> COM RxPDO-Map Outputs Channel 2/Data Out 9
//   SDSM3/SDSM3 Instance <-> MAIN (EtherCAT)/PCM B (EP3174-0002)
//     PlcTask Inputs/GVL_IO.iq_stPressCtrlB.i_EP3174_Ch{1..4} <-> AI Standard Channel {1..4}/Value  (4 links)
//   SDSM3/SDSM3 Instance <-> MAIN (EtherCAT)/PCM B (EP4374-0002)
//     PlcTask Inputs/GVL_IO.iq_stPressCtrlB.i_EP4374_Ch1 <-> AI Inputs Channel 1/Value
//     PlcTask Inputs/GVL_IO.iq_stPressCtrlB.i_EP4374_Ch2 <-> AI Inputs Channel 2/Value
//     PlcTask Outputs/GVL_IO.iq_stPressCtrlB.q_EP4374_Ch3 <-> AO Outputs Channel 3/Analog output
//     PlcTask Outputs/GVL_IO.iq_stPressCtrlB.q_EP4374_Ch4 <-> AO Outputs Channel 4/Analog output
//   SDSM3/SDSM3 Instance <-> MAIN (EtherCAT)/PCM B (EP6002-0002)
//     PlcTask Inputs/GVL_IO.iq_stPressCtrlB.stComIn_EP6002P1/D[0] <-> COM TxPDO-Map Inputs Channel 1/Data In 0
//     PlcTask Inputs/GVL_IO.iq_stPressCtrlB.stComIn_EP6002P1/D[10] <-> COM TxPDO-Map Inputs Channel 1/Data In 10
//     PlcTask Inputs/GVL_IO.iq_stPressCtrlB.stComIn_EP6002P1/D[11] <-> COM TxPDO-Map Inputs Channel 1/Data In 11
//     PlcTask Inputs/GVL_IO.iq_stPressCtrlB.stComIn_EP6002P1/D[12] <-> COM TxPDO-Map Inputs Channel 1/Data In 12
//     PlcTask Inputs/GVL_IO.iq_stPressCtrlB.stComIn_EP6002P1/D[13] <-> COM TxPDO-Map Inputs Channel 1/Data In 13
//     PlcTask Inputs/GVL_IO.iq_stPressCtrlB.stComIn_EP6002P1/D[14] <-> COM TxPDO-Map Inputs Channel 1/Data In 14
//     PlcTask Inputs/GVL_IO.iq_stPressCtrlB.stComIn_EP6002P1/D[15] <-> COM TxPDO-Map Inputs Channel 1/Data In 15
//     PlcTask Inputs/GVL_IO.iq_stPressCtrlB.stComIn_EP6002P1/D[16] <-> COM TxPDO-Map Inputs Channel 1/Data In 16
//     PlcTask Inputs/GVL_IO.iq_stPressCtrlB.stComIn_EP6002P1/D[17] <-> COM TxPDO-Map Inputs Channel 1/Data In 17
//     PlcTask Inputs/GVL_IO.iq_stPressCtrlB.stComIn_EP6002P1/D[18] <-> COM TxPDO-Map Inputs Channel 1/Data In 18
//     PlcTask Inputs/GVL_IO.iq_stPressCtrlB.stComIn_EP6002P1/D[19] <-> COM TxPDO-Map Inputs Channel 1/Data In 19
//     PlcTask Inputs/GVL_IO.iq_stPressCtrlB.stComIn_EP6002P1/D[1] <-> COM TxPDO-Map Inputs Channel 1/Data In 1
//     PlcTask Inputs/GVL_IO.iq_stPressCtrlB.stComIn_EP6002P1/D[20] <-> COM TxPDO-Map Inputs Channel 1/Data In 20
//     PlcTask Inputs/GVL_IO.iq_stPressCtrlB.stComIn_EP6002P1/D[21] <-> COM TxPDO-Map Inputs Channel 1/Data In 21
//     PlcTask Inputs/GVL_IO.iq_stPressCtrlB.stComIn_EP6002P1/D[2] <-> COM TxPDO-Map Inputs Channel 1/Data In 2
//     PlcTask Inputs/GVL_IO.iq_stPressCtrlB.stComIn_EP6002P1/D[3] <-> COM TxPDO-Map Inputs Channel 1/Data In 3
//     PlcTask Inputs/GVL_IO.iq_stPressCtrlB.stComIn_EP6002P1/D[4] <-> COM TxPDO-Map Inputs Channel 1/Data In 4
//     PlcTask Inputs/GVL_IO.iq_stPressCtrlB.stComIn_EP6002P1/D[5] <-> COM TxPDO-Map Inputs Channel 1/Data In 5
//     PlcTask Inputs/GVL_IO.iq_stPressCtrlB.stComIn_EP6002P1/D[6] <-> COM TxPDO-Map Inputs Channel 1/Data In 6
//     PlcTask Inputs/GVL_IO.iq_stPressCtrlB.stComIn_EP6002P1/D[7] <-> COM TxPDO-Map Inputs Channel 1/Data In 7
//     PlcTask Inputs/GVL_IO.iq_stPressCtrlB.stComIn_EP6002P1/D[8] <-> COM TxPDO-Map Inputs Channel 1/Data In 8
//     PlcTask Inputs/GVL_IO.iq_stPressCtrlB.stComIn_EP6002P1/D[9] <-> COM TxPDO-Map Inputs Channel 1/Data In 9
//     PlcTask Inputs/GVL_IO.iq_stPressCtrlB.stComIn_EP6002P2/D[0] <-> COM TxPDO-Map Inputs Channel 2/Data In 0
//     PlcTask Inputs/GVL_IO.iq_stPressCtrlB.stComIn_EP6002P2/D[10] <-> COM TxPDO-Map Inputs Channel 2/Data In 10
//     PlcTask Inputs/GVL_IO.iq_stPressCtrlB.stComIn_EP6002P2/D[11] <-> COM TxPDO-Map Inputs Channel 2/Data In 11
//     PlcTask Inputs/GVL_IO.iq_stPressCtrlB.stComIn_EP6002P2/D[12] <-> COM TxPDO-Map Inputs Channel 2/Data In 12
//     PlcTask Inputs/GVL_IO.iq_stPressCtrlB.stComIn_EP6002P2/D[13] <-> COM TxPDO-Map Inputs Channel 2/Data In 13
//     PlcTask Inputs/GVL_IO.iq_stPressCtrlB.stComIn_EP6002P2/D[14] <-> COM TxPDO-Map Inputs Channel 2/Data In 14
//     PlcTask Inputs/GVL_IO.iq_stPressCtrlB.stComIn_EP6002P2/D[15] <-> COM TxPDO-Map Inputs Channel 2/Data In 15
//     PlcTask Inputs/GVL_IO.iq_stPressCtrlB.stComIn_EP6002P2/D[16] <-> COM TxPDO-Map Inputs Channel 2/Data In 16
//     PlcTask Inputs/GVL_IO.iq_stPressCtrlB.stComIn_EP6002P2/D[17] <-> COM TxPDO-Map Inputs Channel 2/Data In 17
//     PlcTask Inputs/GVL_IO.iq_stPressCtrlB.stComIn_EP6002P2/D[18] <-> COM TxPDO-Map Inputs Channel 2/Data In 18
//     PlcTask Inputs/GVL_IO.iq_stPressCtrlB.stComIn_EP6002P2/D[19] <-> COM TxPDO-Map Inputs Channel 2/Data In 19
//     PlcTask Inputs/GVL_IO.iq_stPressCtrlB.stComIn_EP6002P2/D[1] <-> COM TxPDO-Map Inputs Channel 2/Data In 1
//     PlcTask Inputs/GVL_IO.iq_stPressCtrlB.stComIn_EP6002P2/D[20] <-> COM TxPDO-Map Inputs Channel 2/Data In 20
//     PlcTask Inputs/GVL_IO.iq_stPressCtrlB.stComIn_EP6002P2/D[21] <-> COM TxPDO-Map Inputs Channel 2/Data In 21
//     PlcTask Inputs/GVL_IO.iq_stPressCtrlB.stComIn_EP6002P2/D[2] <-> COM TxPDO-Map Inputs Channel 2/Data In 2
//     PlcTask Inputs/GVL_IO.iq_stPressCtrlB.stComIn_EP6002P2/D[3] <-> COM TxPDO-Map Inputs Channel 2/Data In 3
//     PlcTask Inputs/GVL_IO.iq_stPressCtrlB.stComIn_EP6002P2/D[4] <-> COM TxPDO-Map Inputs Channel 2/Data In 4
//     PlcTask Inputs/GVL_IO.iq_stPressCtrlB.stComIn_EP6002P2/D[5] <-> COM TxPDO-Map Inputs Channel 2/Data In 5
//     PlcTask Inputs/GVL_IO.iq_stPressCtrlB.stComIn_EP6002P2/D[6] <-> COM TxPDO-Map Inputs Channel 2/Data In 6
//     PlcTask Inputs/GVL_IO.iq_stPressCtrlB.stComIn_EP6002P2/D[7] <-> COM TxPDO-Map Inputs Channel 2/Data In 7
//     PlcTask Inputs/GVL_IO.iq_stPressCtrlB.stComIn_EP6002P2/D[8] <-> COM TxPDO-Map Inputs Channel 2/Data In 8
//     PlcTask Inputs/GVL_IO.iq_stPressCtrlB.stComIn_EP6002P2/D[9] <-> COM TxPDO-Map Inputs Channel 2/Data In 9
//     PlcTask Inputs/GVL_IO.iq_stPressCtrlB.stComIn_EP6002P1/Status <-> COM TxPDO-Map Inputs Channel 1/Status
//     PlcTask Inputs/GVL_IO.iq_stPressCtrlB.stComIn_EP6002P2/Status <-> COM TxPDO-Map Inputs Channel 2/Status
//     PlcTask Outputs/GVL_IO.iq_stPressCtrlB.stComOut_EP6002P1/Ctrl <-> COM RxPDO-Map Outputs Channel 1/Ctrl
//     PlcTask Outputs/GVL_IO.iq_stPressCtrlB.stComOut_EP6002P2/Ctrl <-> COM RxPDO-Map Outputs Channel 2/Ctrl
//     PlcTask Outputs/GVL_IO.iq_stPressCtrlB.stComOut_EP6002P1/D[0] <-> COM RxPDO-Map Outputs Channel 1/Data Out 0
//     PlcTask Outputs/GVL_IO.iq_stPressCtrlB.stComOut_EP6002P1/D[10] <-> COM RxPDO-Map Outputs Channel 1/Data Out 10
//     PlcTask Outputs/GVL_IO.iq_stPressCtrlB.stComOut_EP6002P1/D[11] <-> COM RxPDO-Map Outputs Channel 1/Data Out 11
//     PlcTask Outputs/GVL_IO.iq_stPressCtrlB.stComOut_EP6002P1/D[12] <-> COM RxPDO-Map Outputs Channel 1/Data Out 12
//     PlcTask Outputs/GVL_IO.iq_stPressCtrlB.stComOut_EP6002P1/D[13] <-> COM RxPDO-Map Outputs Channel 1/Data Out 13
//     PlcTask Outputs/GVL_IO.iq_stPressCtrlB.stComOut_EP6002P1/D[14] <-> COM RxPDO-Map Outputs Channel 1/Data Out 14
//     PlcTask Outputs/GVL_IO.iq_stPressCtrlB.stComOut_EP6002P1/D[15] <-> COM RxPDO-Map Outputs Channel 1/Data Out 15
//     PlcTask Outputs/GVL_IO.iq_stPressCtrlB.stComOut_EP6002P1/D[16] <-> COM RxPDO-Map Outputs Channel 1/Data Out 16
//     PlcTask Outputs/GVL_IO.iq_stPressCtrlB.stComOut_EP6002P1/D[17] <-> COM RxPDO-Map Outputs Channel 1/Data Out 17
//     PlcTask Outputs/GVL_IO.iq_stPressCtrlB.stComOut_EP6002P1/D[18] <-> COM RxPDO-Map Outputs Channel 1/Data Out 18
//     PlcTask Outputs/GVL_IO.iq_stPressCtrlB.stComOut_EP6002P1/D[19] <-> COM RxPDO-Map Outputs Channel 1/Data Out 19
//     PlcTask Outputs/GVL_IO.iq_stPressCtrlB.stComOut_EP6002P1/D[1] <-> COM RxPDO-Map Outputs Channel 1/Data Out 1
//     PlcTask Outputs/GVL_IO.iq_stPressCtrlB.stComOut_EP6002P1/D[20] <-> COM RxPDO-Map Outputs Channel 1/Data Out 20
//     PlcTask Outputs/GVL_IO.iq_stPressCtrlB.stComOut_EP6002P1/D[21] <-> COM RxPDO-Map Outputs Channel 1/Data Out 21
//     PlcTask Outputs/GVL_IO.iq_stPressCtrlB.stComOut_EP6002P1/D[2] <-> COM RxPDO-Map Outputs Channel 1/Data Out 2
//     PlcTask Outputs/GVL_IO.iq_stPressCtrlB.stComOut_EP6002P1/D[3] <-> COM RxPDO-Map Outputs Channel 1/Data Out 3
//     PlcTask Outputs/GVL_IO.iq_stPressCtrlB.stComOut_EP6002P1/D[4] <-> COM RxPDO-Map Outputs Channel 1/Data Out 4
//     PlcTask Outputs/GVL_IO.iq_stPressCtrlB.stComOut_EP6002P1/D[5] <-> COM RxPDO-Map Outputs Channel 1/Data Out 5
//     PlcTask Outputs/GVL_IO.iq_stPressCtrlB.stComOut_EP6002P1/D[6] <-> COM RxPDO-Map Outputs Channel 1/Data Out 6
//     PlcTask Outputs/GVL_IO.iq_stPressCtrlB.stComOut_EP6002P1/D[7] <-> COM RxPDO-Map Outputs Channel 1/Data Out 7
//     PlcTask Outputs/GVL_IO.iq_stPressCtrlB.stComOut_EP6002P1/D[8] <-> COM RxPDO-Map Outputs Channel 1/Data Out 8
//     PlcTask Outputs/GVL_IO.iq_stPressCtrlB.stComOut_EP6002P1/D[9] <-> COM RxPDO-Map Outputs Channel 1/Data Out 9
//     PlcTask Outputs/GVL_IO.iq_stPressCtrlB.stComOut_EP6002P2/D[0] <-> COM RxPDO-Map Outputs Channel 2/Data Out 0
//     PlcTask Outputs/GVL_IO.iq_stPressCtrlB.stComOut_EP6002P2/D[10] <-> COM RxPDO-Map Outputs Channel 2/Data Out 10
//     PlcTask Outputs/GVL_IO.iq_stPressCtrlB.stComOut_EP6002P2/D[11] <-> COM RxPDO-Map Outputs Channel 2/Data Out 11
//     PlcTask Outputs/GVL_IO.iq_stPressCtrlB.stComOut_EP6002P2/D[12] <-> COM RxPDO-Map Outputs Channel 2/Data Out 12
//     PlcTask Outputs/GVL_IO.iq_stPressCtrlB.stComOut_EP6002P2/D[13] <-> COM RxPDO-Map Outputs Channel 2/Data Out 13
//     PlcTask Outputs/GVL_IO.iq_stPressCtrlB.stComOut_EP6002P2/D[14] <-> COM RxPDO-Map Outputs Channel 2/Data Out 14
//     PlcTask Outputs/GVL_IO.iq_stPressCtrlB.stComOut_EP6002P2/D[15] <-> COM RxPDO-Map Outputs Channel 2/Data Out 15
//     PlcTask Outputs/GVL_IO.iq_stPressCtrlB.stComOut_EP6002P2/D[16] <-> COM RxPDO-Map Outputs Channel 2/Data Out 16
//     PlcTask Outputs/GVL_IO.iq_stPressCtrlB.stComOut_EP6002P2/D[17] <-> COM RxPDO-Map Outputs Channel 2/Data Out 17
//     PlcTask Outputs/GVL_IO.iq_stPressCtrlB.stComOut_EP6002P2/D[18] <-> COM RxPDO-Map Outputs Channel 2/Data Out 18
//     PlcTask Outputs/GVL_IO.iq_stPressCtrlB.stComOut_EP6002P2/D[19] <-> COM RxPDO-Map Outputs Channel 2/Data Out 19
//     PlcTask Outputs/GVL_IO.iq_stPressCtrlB.stComOut_EP6002P2/D[1] <-> COM RxPDO-Map Outputs Channel 2/Data Out 1
//     PlcTask Outputs/GVL_IO.iq_stPressCtrlB.stComOut_EP6002P2/D[20] <-> COM RxPDO-Map Outputs Channel 2/Data Out 20
//     PlcTask Outputs/GVL_IO.iq_stPressCtrlB.stComOut_EP6002P2/D[21] <-> COM RxPDO-Map Outputs Channel 2/Data Out 21
//     PlcTask Outputs/GVL_IO.iq_stPressCtrlB.stComOut_EP6002P2/D[2] <-> COM RxPDO-Map Outputs Channel 2/Data Out 2
//     PlcTask Outputs/GVL_IO.iq_stPressCtrlB.stComOut_EP6002P2/D[3] <-> COM RxPDO-Map Outputs Channel 2/Data Out 3
//     PlcTask Outputs/GVL_IO.iq_stPressCtrlB.stComOut_EP6002P2/D[4] <-> COM RxPDO-Map Outputs Channel 2/Data Out 4
//     PlcTask Outputs/GVL_IO.iq_stPressCtrlB.stComOut_EP6002P2/D[5] <-> COM RxPDO-Map Outputs Channel 2/Data Out 5
//     PlcTask Outputs/GVL_IO.iq_stPressCtrlB.stComOut_EP6002P2/D[6] <-> COM RxPDO-Map Outputs Channel 2/Data Out 6
//     PlcTask Outputs/GVL_IO.iq_stPressCtrlB.stComOut_EP6002P2/D[7] <-> COM RxPDO-Map Outputs Channel 2/Data Out 7
//     PlcTask Outputs/GVL_IO.iq_stPressCtrlB.stComOut_EP6002P2/D[8] <-> COM RxPDO-Map Outputs Channel 2/Data Out 8
//     PlcTask Outputs/GVL_IO.iq_stPressCtrlB.stComOut_EP6002P2/D[9] <-> COM RxPDO-Map Outputs Channel 2/Data Out 9
//   SDSM3/SDSM3 Instance <-> NC-Task 1 SAF/Axes/ALI_PropValve
//     PlcTask Inputs/GVL_Devices.stALI.stPropVlv.stAxis.NcToPlc <-> Outputs/ToPlc
//     PlcTask Outputs/GVL_Devices.stALI.stPropVlv.stAxis.PlcToNc <-> Inputs/FromPlc
//   SDSM3/SDSM3 Instance <-> NC-Task 1 SAF/Axes/ALI_X
//     PlcTask Inputs/GVL_Devices.stALI.axisX.stAxis.NcToPlc <-> Outputs/ToPlc
//     PlcTask Outputs/GVL_Devices.stALI.axisX.stAxis.PlcToNc <-> Inputs/FromPlc
//   SDSM3/SDSM3 Instance <-> NC-Task 1 SAF/Axes/ALI_Y
//     PlcTask Inputs/GVL_Devices.stALI.axisY.stAxis.NcToPlc <-> Outputs/ToPlc
//     PlcTask Outputs/GVL_Devices.stALI.axisY.stAxis.PlcToNc <-> Inputs/FromPlc
//   SDSM3/SDSM3 Instance <-> NC-Task 1 SAF/Axes/ALI_Z
//     PlcTask Inputs/GVL_Devices.stALI.axisZ.stAxis.NcToPlc <-> Outputs/ToPlc
//     PlcTask Outputs/GVL_Devices.stALI.axisZ.stAxis.PlcToNc <-> Inputs/FromPlc

CONFIGURATION SDSM3
    RESOURCE PLC ON TwinCAT3
        TASK PlcTask(INTERVAL := T#10ms, PRIORITY := 20);
        PROGRAM MAIN WITH PlcTask : MAIN;
    END_RESOURCE
END_CONFIGURATION

// ---- DUTs/ALI/E_CTRL_MODE.TcDUT
{attribute 'qualified_only'}
{attribute 'strict'}
TYPE E_CTRL_MODE :
(
	Init := 0,
	Run	:= 10,
	Hold	:= 20,
	Error	:= 9000
);
END_TYPE

// ---- DUTs/ALI/HMI_PropValveCtrlState.TcDUT
{attribute 'qualified_only'}
(* Maps to an EPICS MBBI/O *)
TYPE HMI_PropValveCtrlState :
(
	Manual := 0,
	Pressure := 1,
	Hold := 2
) WORD;
END_TYPE

// ---- DUTs/ALI/ST_ALI.TcDUT
TYPE ST_ALI EXTENDS ST_ALIIO:
STRUCT
	(* Aerodynamic Lens Injector *)

	(* Manipulator *)
	axisX	:	ST_ManipAxis;
	axisY	:	ST_ManipAxis;
	axisZ	:	ST_ManipAxis;
	
	(* Vacuum gauges *)
	//925
	stNozzleBoxVG	: ST_VG;
	//925
	stSkimmerVG	: ST_VG;
	//722
	stRelaxVG	: ST_VG := (rFULL_SCALE:=10);
	
	(* Butterfly valve pressure controller *)
	stPropVlv	:	ST_PropValveMKS253;
	
	(* PropValve Pressure Controller *)
	//stPressCtrl	:	ST_PressureController;
	
	
END_STRUCT
END_TYPE

// ---- DUTs/ALI/ST_ManipAxis.TcDUT
TYPE ST_ManipAxis :
STRUCT

(* Controls *)
xEnable	:	BOOL := TRUE;
rReqAbsPos	:	REAL;
rReqRelPos	:	REAL;
xStart	:	BOOL;
xStop	:	BOOL;
wMode	:	E_AxisMoveMode;
//EPICS motor status
uiMsta	:	UINT;
//EPICS Position readback
rActPos	:	REAL;
//Axis enabled readback
xEnabled	:	BOOL;
//EPICS High Limit Switch (NO)
xHLS	:	BOOL;
//EPICS Low Limit Switch (NO)
xLLS	:	BOOL;
//EPICS MOVN
xMovn	:	BOOL;
//EPICS DMOV
xDmov	:	BOOL;
//EPICS Reset
xReset	:	BOOL;
	
(* Axis motor *)
stAxis	:	AXIS_REF;
lrVelocity	:	LREAL	:=1; //mm/s

eState	:	E_AxisMotionState;

xHiLS	AT %I* :	BOOL;
xLoLS	AT %I* :	BOOL;

END_STRUCT
END_TYPE

// ---- DUTs/ALI/ST_PIDParams.TcDUT
TYPE ST_PIDParams :
STRUCT
	fCtrlCycleTime : LREAL; (* controller cycle time in seconds [s] *)
    fKp            : LREAL; (* proportional gain Kp (P) *)
    fTn            : LREAL; (* integral gain Tn (I) [s] *)
    fTv            : LREAL; (* derivative gain Tv (D-T1) [s] *)
    fTd            : LREAL; (* derivative damping time Td (D-T1) [s] *)
	fUpperLim		: 	LREAL; (* upper controller output range limit of PID block *)
	fLowerLim		:	LREAL; (* lower controller output range limit of PID block *)
END_STRUCT
END_TYPE

// ---- DUTs/ALI/ST_PressureController.TcDUT
TYPE ST_PressureController :
STRUCT
	(* Intent of this structure is to provide generic variables
	for a pressure controller. It is meant to be extended by 
	the hardware IO variables into a specific structure. *)
	
	//Controls
	//Pressure setpoint
	i_rPressSP	:	REAL;
	//Pressure readback
	i_rPressRB	:	REAL;
	//Controller deadband
	rDeadband	:	REAL;
	//Actuator percentage open setpoint 0-100%
	i_iPercOpenSP	:	INT;
	//Acuator percentage open readback
	q_iPercOpen	:	INT;
	//Controller Mode
	i_eCntlMode	:	E_CTRL_MODE;
	//PID Parameters
	stPIDParams :	ST_PIDParams := (
		fKp := 1,
		fTn := 1,
		fUpperLim := 1,
		fLowerLim := -1,
		fCtrlCycleTime := 0.01
	);
	
END_STRUCT
END_TYPE

// ---- DUTs/ALI/ST_PropValveMKS253.TcDUT
TYPE ST_PropValveMKS253 EXTENDS ST_PressureController:
STRUCT
	
	(* Prop valve structure, open is considered to be the higher axis position *)
	(* Note: The wiring (if using the dongle from the ALI schematic is such that the 
	stepper driver must be inverted to make the increasing counter value correspond to a more open valve. *)
	
	//EPICS Enable Switch
	xEnable	:	BOOL;
	//EPICS Enable Control;
	xEnabled	:	BOOL;
	//Valve interlock
	xInterlock	:	BOOL;
	//PropValve Control State Control
	ePVCtrlStateReq : HMI_PropValveCtrlState;
	//PropValve Control State Readback
	ePVCtrlState : HMI_PropValveCtrlState;
	//NC Axis Ref
	stAxis	:	AXIS_REF;
	//Physical limit switches
	i_HLS	AT %I*	:	BOOL; //Open
	i_LLS	AT %I*	:	BOOL; // Closed
	//Open EPICS LS
	xHLS	:	BOOL;
	//Close EPICS LS
	xLLS	:	BOOL;
	//Top speed for the valve
	lrMaxSpeed	:	LREAL := 100; //deg/sec
END_STRUCT
END_TYPE

// ---- DUTs/Bronkhorst/ST_BhElFlow.TcDUT
TYPE ST_BhElFlow :
STRUCT
	eFlowUnit	:	E_BHElFlowUnit;
	i_udiUnit	:	UDINT;
	i_rFlow	:	REAL;
END_STRUCT
END_TYPE

// ---- DUTs/Bronkhorst/ST_BhFMControl.TcDUT
TYPE ST_BhFMControl :
STRUCT
	xReset	:	BOOL;
END_STRUCT
END_TYPE

// ---- DUTs/Bronkhorst/ST_BhFMStatus.TcDUT
TYPE ST_BhFMStatus :
STRUCT
	
uiFlowPercentageRaw	:	UINT;
	rFlowPercentage	: REAL;
	rFlow	:	REAL;
	xOoR	:	BOOL; // Out of range above
xFlowValid	:	BOOL;
	sReply	:	STRING;
	iState	:	INT;

END_STRUCT
END_TYPE

// ---- DUTs/E_AxisMotionState.TcDUT
TYPE E_AxisMotionState :
(
	Init := 10,
	MoveEnabled := 3000,
	Error := 9000
);
END_TYPE

// ---- DUTs/IO_Structs/ST_ALIIO.TcDUT
TYPE ST_ALIIO EXTENDS ST_M3DeviceBaseIO :
STRUCT
	//EP7041
	//EP7041
	//EP7041
	//EP5101
	//EP3174 Vacuum Gauges, misc analog
	i_EP3174_Ch1	AT	%I*	:	INT;
	i_EP3174_Ch2	AT	%I*	:	INT;
	i_EP3174_Ch3	AT	%I*	:	INT;
	i_EP3174_Ch4	AT	%I*	:	INT;
	//EP7041 - Prop valve
	
	
END_STRUCT
END_TYPE

// ---- DUTs/IO_Structs/ST_M2SelectorIO.TcDUT
TYPE ST_M2SelectorIO EXTENDS ST_M3DeviceBaseIO:
STRUCT

	q_EP2338_Ch1	AT	%Q*	:	BOOL;
	q_EP2338_Ch2	AT	%Q*	:	BOOL;
	q_EP2338_Ch3	AT	%Q*	:	BOOL;
	q_EP2338_Ch4	AT	%Q*	:	BOOL;
	
	i_EP2338_Ch5	AT	%I*	:	BOOL;
	i_EP2338_Ch6	AT	%I*	:	BOOL;
	i_EP2338_Ch7	AT	%I*	:	BOOL;
	i_EP2338_Ch8	AT	%I*	:	BOOL;


	stComIn_EP6002P1		AT %I*	:	EL6inData22B (*KL6inData22B*);
	stComOut_EP6002P1		AT %Q*	:	EL6outData22B (*KL6outData22B*);
	
	stComIn_EP6002P2		AT %I*	:	EL6inData22B (*KL6inData22B*);
	stComOut_EP6002P2		AT %Q*	:	EL6outData22B (*KL6outData22B*);
	
END_STRUCT
END_TYPE

// ---- DUTs/IO_Structs/ST_M3SelectorIO.TcDUT
TYPE ST_M3SelectorIO EXTENDS ST_M2SelectorIO:
STRUCT
	
	i_mfmFlow		AT	%I*	:	REAL;
	i_RawUnit		AT %I*	:	UDINT;
	
END_STRUCT
END_TYPE

// ---- DUTs/Sensirion/ST_SensirionFMControl.TcDUT
TYPE ST_SensirionFMControl :
STRUCT
	
xCalMode	:	BOOL;

xReset		:	BOOL;
	

END_STRUCT
END_TYPE

